  MoveC 1133 to (433.16, 156.25, -8.35) mm, rotated rx 180 ry 0 rz -179 deg; joints [11.722, -45.324, 75.106, 22.673, -31.807, -19.546] to (420.46, 168.95, -8.35) mm, rotated rx -180 ry 0 rz -179 deg; joints [11.384, -46.351, 76.909, 21.605, -32.417, -18.486]
  MoveL 1134 to (395.06, 168.95, -8.35) mm, rotated rx -180 ry 0 rz -179 deg; joints [11.539, -48.04, 79.855, 21.171, -33.635, -17.872]
  MoveL 1135 to (318.86, 168.95, -8.35) mm, rotated rx -180 ry 0 rz -179 deg; joints [12.033, -52.857, 88.085, 20.282, -36.974, -16.448]
  MoveC 1136 to (306.16, 156.25, -8.35) mm, rotated rx -180 ry 0 rz -179 deg; joints [12.565, -53.476, 89.123, 20.928, -37.518, -16.874] to (293.46, 168.95, -8.35) mm, rotated rx -180 ry 0 rz -179 deg; joints [12.208, -54.397, 90.66, 20.092, -37.994, -16.081]
  MoveL 1137 to (191.86, 168.95, -8.35) mm, rotated rx -180 ry 0 rz -179 deg; joints [12.967, -60.337, 100.305, 19.72, -41.681, -14.987]
  MoveC 1138 to (179.16, 156.25, -8.35) mm, rotated rx 180 ry 0 rz -179 deg; joints [13.549, -60.904, 101.2, 20.435, -42.142, -15.444] to (166.46, 168.95, -8.35) mm, rotated rx 180 ry 0 rz -179 deg; joints [13.172, -61.782, 102.578, 19.708, -42.513, -14.791]
  MoveL 1139 to (90.26, 168.95, -8.35) mm, rotated rx -180 ry 0 rz -179 deg; joints [13.833, -66.063, 109.12, 19.833, -44.808, -14.353]
  MoveL 1140 to (64.86, 168.95, -8.35) mm, rotated rx -180 ry 0 rz -179 deg; joints [14.069, -67.479, 111.218, 19.925, -45.508, -14.253]
  MoveC 1141 to (61.14, 159.97, -8.35) mm, rotated rx -180 ry 0 rz -179 deg; joints [14.471, -67.568, 111.349, 20.456, -45.647, -14.615] to (52.16, 156.25, -8.35) mm, rotated rx 180 ry 0 rz -179 deg; joints [14.712, -68.017, 112.007, 20.709, -45.903, -14.739]
  MoveL 1142 to (52.16, 156.25, -8.35) mm, rotated rx 180 ry 0 rz -179 deg; joints [14.712, -68.017, 112.007, 20.709, -45.903, -14.739]
  MoveC 1143 to (43.18, 159.97, -8.35) mm, rotated rx -180 ry 0 rz -179 deg; joints [14.649, -68.566, 112.806, 20.539, -46.122, -14.558] to (39.46, 168.95, -8.35) mm, rotated rx -180 ry 0 rz -179 deg; joints [14.314, -68.892, 113.279, 20.041, -46.176, -14.176]
  MoveL 1144 to (14.06, 168.95, -8.35) mm, rotated rx 180 ry 0 rz -179 deg; joints [14.568, -70.305, 115.303, 20.181, -46.812, -14.12]
  MoveL 1145 to (14.06, 16.55, -8.35) mm, rotated rx 180 ry 0 rz -179 deg; joints [20.81, -67.799, 111.688, 28.732, -47.649, -20.27]
  MoveL 1146 to (19.05, 16.55, -8.35) mm, rotated rx -180 ry 0 rz -179 deg; joints [20.739, -67.53, 111.295, 28.697, -47.515, -20.291]
  MoveC 1147 to (19.49, 16.36, -8.35) mm, rotated rx -180 ry 0 rz -179 deg; joints [20.74, -67.503, 111.254, 28.704, -47.504, -20.3] to (19.68, 15.92, -8.35) mm, rotated rx -180 ry 0 rz -179 deg; joints [20.755, -67.484, 111.226, 28.727, -47.501, -20.319]
  MoveL 1148 to (19.68, 15.28, -8.35) mm, rotated rx -180 ry 0 rz -179 deg; joints [20.78, -67.472, 111.208, 28.762, -47.505, -20.344]
  MoveC 1149 to (19.68, 14.83, -8.16) mm, rotated rx 180 ry 0 rz -179 deg; joints [20.798, -67.47, 111.191, 28.791, -47.497, -20.37] to (19.68, 14.65, -7.72) mm, rotated rx 180 ry 0 rz -179 deg; joints [20.805, -67.484, 111.173, 28.814, -47.473, -20.396]
  Set speed (500.0 mm/s)
  MoveL 1150 to (19.68, 14.65, 6) mm, rotated rx -180 ry 0 rz -179 deg; joints [20.805, -68, 110.8, 29.215, -46.695, -20.985]
  MoveL 1151 to (12.15, -16.75, 6) mm, rotated rx -180 ry 0 rz -179 deg; joints [22.145, -67.773, 110.469, 30.97, -47.099, -22.222]
  Set speed (25.4 mm/s)
  MoveL 1152 to (12.15, -16.75, -4.37) mm, rotated rx 180 ry 0 rz -179 deg; joints [22.145, -67.386, 110.753, 30.654, -47.675, -21.756]
  MoveC 1153 to (12.34, -16.75, -4.81) mm, rotated rx -180 ry 0 rz -179 deg; joints [22.142, -67.359, 110.75, 30.639, -47.694, -21.736] to (12.79, -16.75, -5) mm, rotated rx -180 ry 0 rz -179 deg; joints [22.135, -67.328, 110.72, 30.63, -47.693, -21.73]
  Set speed (50.8 mm/s)
  MoveL 1154 to (13.42, -16.75, -5) mm, rotated rx -180 ry 0 rz -179 deg; joints [22.126, -67.294, 110.67, 30.626, -47.675, -21.733]
  MoveC 1155 to (13.87, -16.94, -5) mm, rotated rx -180 ry 0 rz -179 deg; joints [22.126, -67.266, 110.629, 30.633, -47.664, -21.743] to (14.06, -17.39, -5) mm, rotated rx 180 ry 0 rz -179 deg; joints [22.141, -67.247, 110.601, 30.655, -47.662, -21.761]
  MoveL 1156 to (14.06, -169.79, -5) mm, rotated rx -180 ry 0 rz -179 deg; joints [27.82, -63.684, 105.249, 38.496, -48.568, -27.757]
  MoveL 1157 to (471.26, -169.79, -5) mm, rotated rx -180 ry 0 rz -179 deg; joints [21.439, -35.651, 57.394, 46.669, -30.164, -42.505]
  MoveL 1158 to (471.26, -17.39, -5) mm, rotated rx 180 ry 0 rz -179 deg; joints [16.91, -39.664, 64.74, 35.652, -29.935, -31.866]
  MoveL 1159 to (445.86, -17.39, -5) mm, rotated rx -180 ry 0 rz -179 deg; joints [17.133, -41.565, 68.171, 34.541, -31.303, -30.461]
  MoveC 1160 to (433.16, -30.09, -5) mm, rotated rx -180 ry 0 rz -179 deg; joints [17.641, -42.214, 69.335, 34.898, -31.985, -30.611] to (420.46, -17.39, -5) mm, rotated rx -180 ry 0 rz -179 deg; joints [17.363, -43.381, 71.42, 33.631, -32.604, -29.264]
  MoveL 1161 to (395.06, -17.39, -5) mm, rotated rx 180 ry 0 rz -179 deg; joints [17.599, -45.128, 74.514, 32.88, -33.845, -28.231]
  MoveL 1162 to (318.86, -17.39, -5) mm, rotated rx 180 ry 0 rz -179 deg; joints [18.35, -50.044, 83.06, 31.33, -37.261, -25.849]
  MoveC 1163 to (306.16, -30.09, -5) mm, rotated rx 180 ry 0 rz -179 deg; joints [18.901, -50.578, 83.972, 31.885, -37.825, -26.168] to (293.46, -17.39, -5) mm, rotated rx 180 ry 0 rz -179 deg; joints [18.614, -51.599, 85.709, 30.99, -38.311, -25.234]
  MoveL 1164 to (191.86, -17.39, -5) mm, rotated rx -180 ry 0 rz -179 deg; joints [19.757, -57.528, 95.542, 30.252, -42.142, -23.386]
  MoveC 1165 to (179.16, -30.09, -5) mm, rotated rx 180 ry 0 rz -179 deg; joints [20.359, -57.996, 96.299, 30.909, -42.631, -23.772] to (166.46, -17.39, -5) mm, rotated rx -180 ry 0 rz -179 deg; joints [20.065, -58.955, 97.84, 30.193, -43.017, -23.046]
  MoveL 1166 to (90.26, -17.39, -5) mm, rotated rx -180 ry 0 rz -179 deg; joints [21.052, -63.146, 104.423, 30.261, -45.463, -22.255]
  MoveL 1167 to (64.86, -17.39, -5) mm, rotated rx -180 ry 0 rz -179 deg; joints [21.403, -64.521, 106.524, 30.358, -46.223, -22.059]
  MoveC 1168 to (61.14, -26.37, -5) mm, rotated rx -180 ry 0 rz -179 deg; joints [21.794, -64.539, 106.552, 30.855, -46.379, -22.399] to (52.16, -30.09, -5) mm, rotated rx -180 ry 0 rz -179 deg; joints [22.064, -64.945, 107.167, 31.097, -46.661, -22.487]
  MoveL 1169 to (52.16, -30.09, -5) mm, rotated rx -180 ry 0 rz -179 deg; joints [22.064, -64.945, 107.167, 31.097, -46.661, -22.487]
  MoveC 1170 to (43.18, -26.37, -5) mm, rotated rx -180 ry 0 rz -179 deg; joints [22.054, -65.503, 108.008, 30.947, -46.9, -22.279] to (39.46, -17.39, -5) mm, rotated rx -180 ry 0 rz -179 deg; joints [21.766, -65.887, 108.583, 30.49, -46.955, -21.895]
  MoveL 1171 to (14.06, -17.39, -5) mm, rotated rx -180 ry 0 rz -179 deg; joints [22.141, -67.247, 110.601, 30.655, -47.662, -21.761]
  MoveC 1172 to (13.61, -17.2, -5) mm, rotated rx -180 ry 0 rz -179 deg; joints [22.14, -67.275, 110.642, 30.648, -47.673, -21.752] to (13.42, -16.75, -5) mm, rotated rx -180 ry 0 rz -179 deg; joints [22.126, -67.294, 110.67, 30.626, -47.675, -21.733]
  MoveL 1173 to (13.42, -16.12, -5) mm, rotated rx -180 ry 0 rz -179 deg; joints [22.101, -67.307, 110.689, 30.592, -47.671, -21.708]
  MoveC 1174 to (13.42, -15.67, -4.81) mm, rotated rx -180 ry 0 rz -179 deg; joints [22.084, -67.323, 110.698, 30.574, -47.658, -21.698] to (13.42, -15.48, -4.37) mm, rotated rx -180 ry 0 rz -179 deg; joints [22.076, -67.344, 110.692, 30.577, -47.632, -21.711]
  Set speed (500.0 mm/s)
  MoveL 1175 to (13.42, -15.48, 5) mm, rotated rx -180 ry 0 rz -179 deg; joints [22.076, -67.694, 110.436, 30.862, -47.112, -22.131]
  MoveL 1176 to (12.15, -16.75, 5) mm, rotated rx -180 ry 0 rz -179 deg; joints [22.145, -67.736, 110.497, 30.939, -47.154, -22.177]
  Set speed (25.4 mm/s)
  MoveL 1177 to (12.15, -16.75, 1) mm, rotated rx -180 ry 0 rz -179 deg; joints [22.145, -67.587, 110.607, 30.816, -47.376, -21.996]
  MoveL 1178 to (12.15, -16.75, -7.71) mm, rotated rx 180 ry 0 rz -179 deg; joints [22.145, -67.259, 110.843, 30.554, -47.861, -21.607]
  MoveC 1179 to (12.34, -16.75, -8.16) mm, rotated rx -180 ry 0 rz -179 deg; joints [22.142, -67.232, 110.84, 30.539, -47.881, -21.588] to (12.79, -16.75, -8.35) mm, rotated rx 180 ry 0 rz -179 deg; joints [22.135, -67.201, 110.81, 30.531, -47.879, -21.582]
  Set speed (50.8 mm/s)
  MoveL 1180 to (13.42, -16.75, -8.35) mm, rotated rx -180 ry 0 rz -179 deg; joints [22.126, -67.167, 110.76, 30.526, -47.861, -21.584]
  MoveC 1181 to (13.87, -16.94, -8.35) mm, rotated rx 180 ry 0 rz -179 deg; joints [22.126, -67.139, 110.719, 30.533, -47.85, -21.594] to (14.06, -17.39, -8.35) mm, rotated rx -180 ry 0 rz -179 deg; joints [22.141, -67.12, 110.69, 30.555, -47.848, -21.613]
  MoveL 1182 to (14.06, -169.79, -8.35) mm, rotated rx 180 ry 0 rz -179 deg; joints [27.82, -63.565, 105.338, 38.383, -48.731, -27.585]
  MoveL 1183 to (471.26, -169.79, -8.35) mm, rotated rx -180 ry 0 rz -179 deg; joints [21.439, -35.589, 57.514, 46.442, -30.289, -42.242]
  MoveL 1184 to (471.26, -17.39, -8.35) mm, rotated rx -180 ry 0 rz -179 deg; joints [16.91, -39.592, 64.848, 35.471, -30.082, -31.656]
  MoveL 1185 to (445.86, -17.39, -8.35) mm, rotated rx -180 ry 0 rz -179 deg; joints [17.133, -41.488, 68.274, 34.374, -31.452, -30.266]
  MoveC 1186 to (433.16, -30.09, -8.35) mm, rotated rx -180 ry 0 rz -179 deg; joints [17.641, -42.136, 69.438, 34.734, -32.133, -30.418] to (420.46, -17.39, -8.35) mm, rotated rx -180 ry 0 rz -179 deg; joints [17.363, -43.301, 71.52, 33.475, -32.754, -29.08]
  MoveL 1187 to (395.06, -17.39, -8.35) mm, rotated rx -180 ry 0 rz -179 deg; joints [17.599, -45.045, 74.612, 32.734, -33.997, -28.056]
  MoveL 1188 to (318.86, -17.39, -8.35) mm, rotated rx 180 ry 0 rz -179 deg; joints [18.35, -49.952, 83.152, 31.204, -37.419, -25.691]
  MoveC 1189 to (306.16, -30.09, -8.35) mm, rotated rx -180 ry 0 rz -179 deg; joints [18.901, -50.485, 84.064, 31.759, -37.982, -26.009] to (293.46, -17.39, -8.35) mm, rotated rx 180 ry 0 rz -179 deg; joints [18.614, -51.504, 85.799, 30.869, -38.471, -25.08]
  MoveL 1190 to (191.86, -17.39, -8.35) mm, rotated rx 180 ry 0 rz -179 deg; joints [19.757, -57.421, 95.63, 30.144, -42.31, -23.24]
  MoveC 1191 to (179.16, -30.09, -8.35) mm, rotated rx -180 ry 0 rz -179 deg; joints [20.359, -57.889, 96.387, 30.8, -42.799, -23.624] to (166.46, -17.39, -8.35) mm, rotated rx -180 ry 0 rz -179 deg; joints [20.065, -58.846, 97.928, 30.087, -43.187, -22.901]
  MoveL 1192 to (90.26, -17.39, -8.35) mm, rotated rx 180 ry 0 rz -179 deg; joints [21.052, -63.028, 104.512, 30.16, -45.642, -22.11]
  MoveL 1193 to (64.86, -17.39, -8.35) mm, rotated rx 180 ry 0 rz -179 deg; joints [21.403, -64.4, 106.613, 30.257, -46.404, -21.913]
  MoveC 1194 to (61.14, -26.37, -8.35) mm, rotated rx -180 ry 0 rz -179 deg; joints [21.794, -64.418, 106.641, 30.753, -46.559, -22.251] to (52.16, -30.09, -8.35) mm, rotated rx -180 ry 0 rz -179 deg; joints [22.064, -64.823, 107.256, 30.995, -46.841, -22.339]
  MoveL 1195 to (52.16, -30.09, -8.35) mm, rotated rx 180 ry 0 rz -179 deg; joints [22.064, -64.823, 107.256, 30.995, -46.841, -22.339]
  MoveC 1196 to (43.18, -26.37, -8.35) mm, rotated rx 180 ry 0 rz -179 deg; joints [22.054, -65.381, 108.097, 30.846, -47.081, -22.13] to (39.46, -17.39, -8.35) mm, rotated rx -180 ry 0 rz -179 deg; joints [21.766, -65.763, 108.672, 30.39, -47.139, -21.748]
  MoveL 1197 to (14.06, -17.39, -8.35) mm, rotated rx -180 ry 0 rz -179 deg; joints [22.141, -67.12, 110.69, 30.555, -47.848, -21.613]
  MoveC 1198 to (13.61, -17.2, -8.35) mm, rotated rx 180 ry 0 rz -179 deg; joints [22.14, -67.148, 110.731, 30.549, -47.859, -21.603] to (13.42, -16.75, -8.35) mm, rotated rx -180 ry 0 rz -179 deg; joints [22.126, -67.167, 110.76, 30.526, -47.861, -21.584]
  MoveL 1199 to (13.42, -16.12, -8.35) mm, rotated rx 180 ry 0 rz -179 deg; joints [22.101, -67.18, 110.779, 30.492, -47.858, -21.559]
  MoveC 1200 to (13.42, -15.67, -8.16) mm, rotated rx -180 ry 0 rz -179 deg; joints [22.084, -67.196, 110.788, 30.474, -47.845, -21.55] to (13.42, -15.48, -7.72) mm, rotated rx -180 ry 0 rz -179 deg; joints [22.076, -67.217, 110.781, 30.477, -47.819, -21.562]
  Set speed (500.0 mm/s)
  MoveL 1201 to (13.42, -15.48, 6) mm, rotated rx -180 ry 0 rz -179 deg; joints [22.076, -67.731, 110.408, 30.893, -47.056, -22.177]
  MoveL 1202 to (-18.41, -15.48, 6) mm, rotated rx 180 ry 0 rz -179 deg; joints [22.565, -69.442, 112.879, 31.147, -47.892, -22.06]
  Set speed (25.4 mm/s)
  MoveL 1203 to (-18.41, -15.48, -4.36) mm, rotated rx 180 ry 0 rz -179 deg; joints [22.565, -69.043, 113.165, 30.832, -48.478, -21.587]
  MoveC 1204 to (-18.41, -15.67, -4.81) mm, rotated rx -180 ry 0 rz -179 deg; joints [22.572, -69.022, 113.172, 30.828, -48.505, -21.574] to (-18.41, -16.12, -5) mm, rotated rx -180 ry 0 rz -179 deg; joints [22.59, -69.005, 113.163, 30.847, -48.518, -21.583]
  Set speed (50.8 mm/s)
  MoveL 1205 to (-18.41, -16.75, -5) mm, rotated rx -180 ry 0 rz -179 deg; joints [22.615, -68.992, 113.144, 30.88, -48.523, -21.608]
  MoveC 1206 to (-18.6, -17.2, -5) mm, rotated rx -180 ry 0 rz -179 deg; joints [22.636, -68.992, 113.145, 30.906, -48.53, -21.625] to (-19.05, -17.39, -5) mm, rotated rx -180 ry 0 rz -179 deg; joints [22.65, -69.012, 113.174, 30.92, -48.543, -21.631]
  MoveL 1207 to (-39.46, -17.39, -5) mm, rotated rx -180 ry 0 rz -179 deg; joints [22.976, -70.099, 114.729, 31.111, -49.065, -21.574]
  MoveC 1208 to (-52.16, -30.09, -5) mm, rotated rx 180 ry 0 rz -179 deg; joints [23.694, -70.496, 115.292, 31.917, -49.474, -22.034] to (-64.86, -17.39, -5) mm, rotated rx -180 ry 0 rz -179 deg; joints [23.394, -71.449, 116.633, 31.377, -49.692, -21.53]
  MoveL 1209 to (-90.26, -17.39, -5) mm, rotated rx -180 ry 0 rz -179 deg; joints [23.828, -72.8, 118.503, 31.676, -50.294, -21.514]
  MoveL 1210 to (-166.46, -17.39, -5) mm, rotated rx 180 ry 0 rz -179 deg; joints [25.231, -76.869, 123.921, 32.772, -51.951, -21.642]
  MoveC 1211 to (-179.16, -30.09, -5) mm, rotated rx 180 ry 0 rz -179 deg; joints [26.031, -77.238, 124.395, 33.668, -52.338, -22.146] to (-191.86, -17.39, -5) mm, rotated rx 180 ry 0 rz -179 deg; joints [25.735, -78.236, 125.666, 33.205, -52.454, -21.745]
  MoveL 1212 to (-293.46, -17.39, -5) mm, rotated rx -180 ry 0 rz -179 deg; joints [27.963, -83.794, 132.347, 35.308, -54.222, -22.493]
  MoveC 1213 to (-306.16, -30.09, -5) mm, rotated rx 180 ry 0 rz -179 deg; joints [28.862, -84.133, 132.733, 36.308, -54.608, -23.053] to (-318.86, -17.39, -5) mm, rotated rx -180 ry 0 rz -179 deg; joints [28.579, -85.214, 133.944, 35.933, -54.604, -22.773]
  MoveL 1214 to (-395.06, -17.39, -5) mm, rotated rx -180 ry 0 rz -179 deg; joints [30.593, -89.571, 138.561, 38.079, -55.608, -23.872]
  MoveL 1215 to (-420.46, -17.39, -5) mm, rotated rx -180 ry 0 rz -179 deg; joints [31.325, -91.061, 140.04, 38.892, -55.899, -24.335]
  MoveC 1216 to (-433.16, -30.09, -5) mm, rotated rx 180 ry 0 rz -179 deg; joints [32.344, -91.362, 140.333, 40.011, -56.317, -24.964] to (-445.86, -17.39, -5) mm, rotated rx 180 ry 0 rz -179 deg; joints [32.091, -92.572, 141.489, 39.758, -56.169, -24.852]
  MoveL 1217 to (-471.26, -17.39, -5) mm, rotated rx 180 ry 0 rz -179 deg; joints [32.892, -94.107, 142.906, 40.68, -56.42, -25.427]
  MoveL 1218 to (-471.26, -169.79, -5) mm, rotated rx 180 ry 0 rz -179 deg; joints [40.129, -88.033, 136.981, 48.184, -59.858, -29.305]
  MoveL 1219 to (-14.06, -169.79, -5) mm, rotated rx -180 ry 0 rz -179 deg; joints [28.334, -65.125, 107.439, 38.694, -49.392, -27.535]
  MoveL 1220 to (-14.06, -17.39, -5) mm, rotated rx 180 ry 0 rz -179 deg; joints [22.572, -68.747, 112.79, 30.877, -48.413, -21.647]
  MoveL 1221 to (-19.05, -17.39, -5) mm, rotated rx -180 ry 0 rz -179 deg; joints [22.65, -69.012, 113.174, 30.92, -48.543, -21.631]
  MoveC 1222 to (-19.49, -17.2, -5) mm, rotated rx 180 ry 0 rz -179 deg; joints [22.65, -69.04, 113.214, 30.914, -48.554, -21.622] to (-19.68, -16.75, -5) mm, rotated rx -180 ry 0 rz -179 deg; joints [22.635, -69.06, 113.242, 30.892, -48.556, -21.604]
  MoveL 1223 to (-19.68, -16.12, -5) mm, rotated rx 180 ry 0 rz -179 deg; joints [22.61, -69.073, 113.261, 30.858, -48.551, -21.579]
  MoveC 1224 to (-19.68, -15.67, -4.81) mm, rotated rx -180 ry 0 rz -179 deg; joints [22.592, -69.09, 113.27, 30.839, -48.538, -21.57] to (-19.68, -15.48, -4.37) mm, rotated rx -180 ry 0 rz -179 deg; joints [22.584, -69.111, 113.263, 30.843, -48.511, -21.583]
  Set speed (500.0 mm/s)
  MoveL 1225 to (-19.68, -15.48, 5) mm, rotated rx -180 ry 0 rz -179 deg; joints [22.584, -69.472, 113.005, 31.127, -47.981, -22.01]
  MoveL 1226 to (-18.41, -15.48, 5) mm, rotated rx -180 ry 0 rz -179 deg; joints [22.565, -69.404, 112.907, 31.116, -47.948, -22.014]
  Set speed (25.4 mm/s)
  MoveL 1227 to (-18.41, -15.48, 1) mm, rotated rx -180 ry 0 rz -179 deg; joints [22.565, -69.25, 113.019, 30.994, -48.175, -21.831]
  MoveL 1228 to (-18.41, -15.48, -7.72) mm, rotated rx 180 ry 0 rz -179 deg; joints [22.565, -68.913, 113.256, 30.732, -48.668, -21.436]
  MoveC 1229 to (-18.41, -15.67, -8.16) mm, rotated rx -180 ry 0 rz -179 deg; joints [22.572, -68.891, 113.263, 30.728, -48.695, -21.423] to (-18.41, -16.12, -8.35) mm, rotated rx 180 ry 0 rz -179 deg; joints [22.59, -68.875, 113.254, 30.747, -48.708, -21.432]
  Set speed (50.8 mm/s)
  MoveL 1230 to (-18.41, -16.75, -8.35) mm, rotated rx -180 ry 0 rz -179 deg; joints [22.615, -68.861, 113.235, 30.781, -48.712, -21.457]
  MoveC 1231 to (-18.6, -17.2, -8.35) mm, rotated rx 180 ry 0 rz -179 deg; joints [22.636, -68.862, 113.235, 30.806, -48.72, -21.474] to (-19.05, -17.39, -8.35) mm, rotated rx 180 ry 0 rz -179 deg; joints [22.65, -68.882, 113.264, 30.82, -48.733, -21.479]
  MoveL 1232 to (-39.46, -17.39, -8.35) mm, rotated rx 180 ry 0 rz -179 deg; joints [22.976, -69.966, 114.82, 31.011, -49.257, -21.421]
  MoveC 1233 to (-52.16, -30.09, -8.35) mm, rotated rx 180 ry 0 rz -179 deg; joints [23.694, -70.362, 115.384, 31.815, -49.665, -21.878] to (-64.86, -17.39, -8.35) mm, rotated rx -180 ry 0 rz -179 deg; joints [23.394, -71.313, 116.725, 31.277, -49.887, -21.375]
  MoveL 1234 to (-90.26, -17.39, -8.35) mm, rotated rx -180 ry 0 rz -179 deg; joints [23.828, -72.661, 118.596, 31.576, -50.492, -21.356]
  MoveL 1235 to (-166.46, -17.39, -8.35) mm, rotated rx 180 ry 0 rz -179 deg; joints [25.231, -76.72, 124.018, 32.668, -52.158, -21.473]
  MoveC 1236 to (-179.16, -30.09, -8.35) mm, rotated rx 180 ry 0 rz -179 deg; joints [26.031, -77.088, 124.492, 33.563, -52.544, -21.974] to (-191.86, -17.39, -8.35) mm, rotated rx -180 ry 0 rz -179 deg; joints [25.735, -78.083, 125.763, 33.1, -52.664, -21.572]
  MoveL 1237 to (-293.46, -17.39, -8.35) mm, rotated rx 180 ry 0 rz -179 deg; joints [27.963, -83.627, 132.451, 35.196, -54.443, -22.301]
  MoveC 1238 to (-306.16, -30.09, -8.35) mm, rotated rx 180 ry 0 rz -179 deg; joints [28.862, -83.965, 132.837, 36.194, -54.828, -22.856] to (-318.86, -17.39, -8.35) mm, rotated rx -180 ry 0 rz -179 deg; joints [28.579, -85.043, 134.05, 35.818, -54.828, -22.574]
  MoveL 1239 to (-395.06, -17.39, -8.35) mm, rotated rx -180 ry 0 rz -179 deg; joints [30.593, -89.388, 138.674, 37.955, -55.841, -23.653]
  MoveL 1240 to (-420.46, -17.39, -8.35) mm, rotated rx -180 ry 0 rz -179 deg; joints [31.325, -90.874, 140.155, 38.765, -56.134, -24.108]
  MoveC 1241 to (-433.16, -30.09, -8.35) mm, rotated rx -180 ry 0 rz -179 deg; joints [32.344, -91.175, 140.449, 39.882, -56.549, -24.731] to (-445.86, -17.39, -8.35) mm, rotated rx 180 ry 0 rz -179 deg; joints [32.091, -92.382, 141.607, 39.627, -56.406, -24.616]
  MoveL 1242 to (-471.26, -17.39, -8.35) mm, rotated rx -180 ry 0 rz -179 deg; joints [32.892, -93.913, 143.027, 40.545, -56.658, -25.182]
  MoveL 1243 to (-471.26, -169.79, -8.35) mm, rotated rx 180 ry 0 rz -179 deg; joints [40.129, -87.855, 137.091, 48.059, -60.051, -29.057]
  MoveL 1244 to (-14.06, -169.79, -8.35) mm, rotated rx -180 ry 0 rz -179 deg; joints [28.334, -65.003, 107.528, 38.582, -49.557, -27.362]
  MoveL 1245 to (-14.06, -17.39, -8.35) mm, rotated rx -180 ry 0 rz -179 deg; joints [22.572, -68.617, 112.88, 30.777, -48.602, -21.496]
  MoveL 1246 to (-19.05, -17.39, -8.35) mm, rotated rx 180 ry 0 rz -179 deg; joints [22.65, -68.882, 113.264, 30.82, -48.733, -21.479]
  MoveC 1247 to (-19.49, -17.2, -8.35) mm, rotated rx -180 ry 0 rz -179 deg; joints [22.65, -68.91, 113.304, 30.814, -48.744, -21.471] to (-19.68, -16.75, -8.35) mm, rotated rx 180 ry 0 rz -179 deg; joints [22.635, -68.929, 113.332, 30.792, -48.745, -21.453]
  MoveL 1248 to (-19.68, -16.12, -8.35) mm, rotated rx -180 ry 0 rz -179 deg; joints [22.61, -68.942, 113.351, 30.758, -48.741, -21.428]
  MoveC 1249 to (-19.68, -15.67, -8.16) mm, rotated rx -180 ry 0 rz -179 deg; joints [22.592, -68.959, 113.36, 30.74, -48.728, -21.419] to (-19.68, -15.48, -7.72) mm, rotated rx 180 ry 0 rz -179 deg; joints [22.584, -68.98, 113.354, 30.743, -48.701, -21.432]
  Set speed (500.0 mm/s)
  MoveL 1250 to (-19.68, -15.48, 6) mm, rotated rx -180 ry 0 rz -179 deg; joints [22.584, -69.51, 112.977, 31.158, -47.924, -22.056]
  MoveL 1251 to (-13.42, -196.51, 6) mm, rotated rx 180 ry 0 rz -179 deg; joints [29.278, -64.766, 106.007, 40.38, -49.013, -29.154]
  Set speed (25.4 mm/s)
  MoveL 1252 to (-13.42, -196.52, -4.36) mm, rotated rx -180 ry 0 rz -179 deg; joints [29.278, -64.399, 106.288, 40.02, -49.508, -28.602]
  MoveC 1253 to (-13.42, -196.7, -4.81) mm, rotated rx -180 ry 0 rz -179 deg; joints [29.284, -64.377, 106.292, 40.014, -49.53, -28.585] to (-13.42, -197.15, -5) mm, rotated rx 180 ry 0 rz -179 deg; joints [29.3, -64.358, 106.278, 40.029, -49.542, -28.593]
  Set speed (50.8 mm/s)
  MoveL 1254 to (-13.42, -197.78, -5) mm, rotated rx 180 ry 0 rz -179 deg; joints [29.323, -64.341, 106.252, 40.06, -49.546, -28.617]
  MoveC 1255 to (-13.61, -198.23, -5) mm, rotated rx -180 ry 0 rz -179 deg; joints [29.342, -64.338, 106.247, 40.084, -49.554, -28.633] to (-14.06, -198.42, -5) mm, rotated rx 180 ry 0 rz -179 deg; joints [29.357, -64.356, 106.274, 40.096, -49.568, -28.636]
  MoveL 1256 to (-39.46, -198.42, -5) mm, rotated rx 180 ry 0 rz -179 deg; joints [29.85, -65.638, 108.21, 40.307, -50.303, -28.449]
  MoveC 1257 to (-52.16, -211.12, -5) mm, rotated rx -180 ry 0 rz -179 deg; joints [30.557, -65.918, 108.63, 41.036, -50.748, -28.843] to (-64.86, -198.42, -5) mm, rotated rx 180 ry 0 rz -179 deg; joints [30.359, -66.911, 110.105, 40.555, -51.019, -28.294]
  MoveL 1258 to (-90.26, -198.42, -5) mm, rotated rx -180 ry 0 rz -179 deg; joints [30.884, -68.176, 111.961, 40.839, -51.715, -28.171]
  MoveL 1259 to (-166.46, -198.42, -5) mm, rotated rx -180 ry 0 rz -179 deg; joints [32.567, -71.935, 117.309, 41.906, -53.7, -27.981]
  MoveC 1260 to (-179.16, -211.12, -5) mm, rotated rx -180 ry 0 rz -179 deg; joints [33.344, -72.168, 117.633, 42.709, -54.133, -28.405] to (-191.86, -198.42, -5) mm, rotated rx -180 ry 0 rz -179 deg; joints [33.166, -73.179, 119.022, 42.332, -54.328, -27.978]
  MoveL 1261 to (-293.46, -198.42, -5) mm, rotated rx -180 ry 0 rz -179 deg; joints [35.779, -78.138, 125.542, 44.391, -56.695, -28.26]
  MoveC 1262 to (-306.16, -211.12, -5) mm, rotated rx 180 ry 0 rz -179 deg; joints [36.635, -78.319, 125.771, 45.267, -57.137, -28.71] to (-318.86, -198.42, -5) mm, rotated rx 180 ry 0 rz -179 deg; joints [36.491, -79.376, 127.091, 44.997, -57.254, -28.407]
  MoveL 1263 to (-395.06, -198.42, -5) mm, rotated rx -180 ry 0 rz -179 deg; joints [38.787, -83.099, 131.548, 47.039, -58.868, -29.039]
  MoveL 1264 to (-420.46, -198.42, -5) mm, rotated rx 180 ry 0 rz -179 deg; joints [39.609, -84.344, 132.971, 47.798, -59.389, -29.316]
  MoveC 1265 to (-433.16, -211.12, -5) mm, rotated rx 180 ry 0 rz -179 deg; joints [40.554, -84.46, 133.102, 48.744, -59.865, -29.784] to (-445.86, -198.42, -5) mm, rotated rx -180 ry 0 rz -179 deg; joints [40.462, -85.591, 134.361, 48.596, -59.904, -29.627]
  MoveL 1266 to (-471.26, -198.42, -5) mm, rotated rx 180 ry 0 rz -179 deg; joints [41.347, -86.841, 135.719, 49.434, -60.414, -29.973]
  MoveL 1267 to (-471.26, -350.82, -5) mm, rotated rx -180 ry 0 rz -179 deg; joints [47.144, -80.326, 128.256, 55.442, -62.888, -33.491]
  MoveL 1268 to (-14.06, -350.82, -5) mm, rotated rx -180 ry 0 rz -179 deg; joints [34.476, -59.803, 99.193, 47.256, -50.424, -34.581]
  MoveL 1269 to (-14.06, -198.42, -5) mm, rotated rx 180 ry 0 rz -179 deg; joints [29.357, -64.356, 106.274, 40.096, -49.568, -28.636]
  MoveC 1270 to (-13.87, -197.97, -5) mm, rotated rx -180 ry 0 rz -179 deg; joints [29.338, -64.359, 106.279, 40.073, -49.56, -28.621] to (-13.42, -197.78, -5) mm, rotated rx 180 ry 0 rz -179 deg; joints [29.323, -64.341, 106.252, 40.06, -49.546, -28.617]
  MoveL 1271 to (-12.79, -197.78, -5) mm, rotated rx -180 ry 0 rz -179 deg; joints [29.31, -64.309, 106.203, 40.056, -49.527, -28.622]
  MoveC 1272 to (-12.34, -197.78, -4.81) mm, rotated rx 180 ry 0 rz -179 deg; joints [29.302, -64.293, 106.163, 40.059, -49.505, -28.636] to (-12.15, -197.79, -4.37) mm, rotated rx 180 ry 0 rz -179 deg; joints [29.298, -64.299, 106.137, 40.073, -49.478, -28.661]
  Set speed (500.0 mm/s)
  MoveL 1273 to (-12.15, -197.78, 5) mm, rotated rx 180 ry 0 rz -179 deg; joints [29.298, -64.631, 105.884, 40.398, -49.032, -29.159]
  MoveL 1274 to (-13.42, -196.52, 5) mm, rotated rx 180 ry 0 rz -179 deg; joints [29.278, -64.731, 106.035, 40.345, -49.061, -29.1]
  Set speed (25.4 mm/s)
  MoveL 1275 to (-13.42, -196.51, 1) mm, rotated rx -180 ry 0 rz -179 deg; joints [29.278, -64.59, 106.144, 40.205, -49.251, -28.886]
  MoveL 1276 to (-13.42, -196.51, -7.72) mm, rotated rx 180 ry 0 rz -179 deg; joints [29.278, -64.278, 106.376, 39.906, -49.668, -28.425]
  MoveC 1277 to (-13.42, -196.7, -8.16) mm, rotated rx -180 ry 0 rz -179 deg; joints [29.284, -64.257, 106.38, 39.9, -49.691, -28.409] to (-13.42, -197.15, -8.35) mm, rotated rx 180 ry 0 rz -179 deg; joints [29.3, -64.238, 106.367, 39.915, -49.702, -28.416]
  Set speed (50.8 mm/s)
  MoveL 1278 to (-13.42, -197.78, -8.35) mm, rotated rx -180 ry 0 rz -179 deg; joints [29.323, -64.221, 106.34, 39.946, -49.706, -28.441]
  MoveC 1279 to (-13.61, -198.23, -8.35) mm, rotated rx 180 ry 0 rz -179 deg; joints [29.342, -64.218, 106.336, 39.969, -49.714, -28.457] to (-14.06, -198.42, -8.35) mm, rotated rx -180 ry 0 rz -179 deg; joints [29.357, -64.236, 106.363, 39.982, -49.728, -28.46]
  MoveL 1280 to (-39.46, -198.42, -8.35) mm, rotated rx -180 ry 0 rz -179 deg; joints [29.85, -65.515, 108.299, 40.193, -50.465, -28.271]
  MoveC 1281 to (-52.16, -211.12, -8.35) mm, rotated rx 180 ry 0 rz -179 deg; joints [30.557, -65.795, 108.719, 40.922, -50.909, -28.663] to (-64.86, -198.42, -8.35) mm, rotated rx 180 ry 0 rz -179 deg; joints [30.359, -66.785, 110.194, 40.442, -51.182, -28.115]
  MoveL 1282 to (-90.26, -198.42, -8.35) mm, rotated rx -180 ry 0 rz -179 deg; joints [30.884, -68.047, 112.051, 40.727, -51.881, -27.989]
  MoveL 1283 to (-166.46, -198.42, -8.35) mm, rotated rx -180 ry 0 rz -179 deg; joints [32.567, -71.798, 117.402, 41.794, -53.871, -27.792]
  MoveC 1284 to (-179.16, -211.12, -8.35) mm, rotated rx -180 ry 0 rz -179 deg; joints [33.344, -72.03, 117.725, 42.596, -54.303, -28.213] to (-191.86, -198.42, -8.35) mm, rotated rx -180 ry 0 rz -179 deg; joints [33.166, -73.039, 119.115, 42.219, -54.501, -27.785]
  MoveL 1285 to (-293.46, -198.42, -8.35) mm, rotated rx -180 ry 0 rz -179 deg; joints [35.779, -77.985, 125.639, 44.277, -56.874, -28.052]
  MoveC 1286 to (-306.16, -211.12, -8.35) mm, rotated rx 180 ry 0 rz -179 deg; joints [36.635, -78.166, 125.868, 45.153, -57.314, -28.499] to (-318.86, -198.42, -8.35) mm, rotated rx -180 ry 0 rz -179 deg; joints [36.491, -79.221, 127.19, 44.882, -57.434, -28.194]
  MoveL 1287 to (-395.06, -198.42, -8.35) mm, rotated rx -180 ry 0 rz -179 deg; joints [38.787, -82.934, 131.652, 46.921, -59.051, -28.81]
  MoveL 1288 to (-420.46, -198.42, -8.35) mm, rotated rx -180 ry 0 rz -179 deg; joints [39.609, -84.175, 133.076, 47.678, -59.573, -29.081]
  MoveC 1289 to (-433.16, -211.12, -8.35) mm, rotated rx -180 ry 0 rz -179 deg; joints [40.554, -84.291, 133.207, 48.625, -60.045, -29.547] to (-445.86, -198.42, -8.35) mm, rotated rx -180 ry 0 rz -179 deg; joints [40.462, -85.419, 134.468, 48.475, -60.088, -29.386]
  MoveL 1290 to (-471.26, -198.42, -8.35) mm, rotated rx -180 ry 0 rz -179 deg; joints [41.347, -86.666, 135.827, 49.312, -60.599, -29.726]
  MoveL 1291 to (-471.26, -350.82, -8.35) mm, rotated rx -180 ry 0 rz -179 deg; joints [47.144, -80.168, 128.356, 55.334, -63.035, -33.253]
  MoveL 1292 to (-14.06, -350.82, -8.35) mm, rotated rx -180 ry 0 rz -179 deg; joints [34.476, -59.692, 99.282, 47.136, -50.559, -34.392]
  MoveL 1293 to (-14.06, -198.42, -8.35) mm, rotated rx -180 ry 0 rz -179 deg; joints [29.357, -64.236, 106.363, 39.982, -49.728, -28.46]
  MoveC 1294 to (-13.87, -197.97, -8.35) mm, rotated rx 180 ry 0 rz -179 deg; joints [29.338, -64.238, 106.367, 39.959, -49.72, -28.444] to (-13.42, -197.78, -8.35) mm, rotated rx -180 ry 0 rz -179 deg; joints [29.323, -64.221, 106.34, 39.946, -49.706, -28.441]
  MoveL 1295 to (-12.79, -197.78, -8.35) mm, rotated rx 180 ry 0 rz -179 deg; joints [29.31, -64.189, 106.291, 39.941, -49.687, -28.446]
  MoveC 1296 to (-12.34, -197.78, -8.16) mm, rotated rx 180 ry 0 rz -179 deg; joints [29.302, -64.173, 106.252, 39.944, -49.665, -28.459] to (-12.15, -197.78, -7.72) mm, rotated rx -180 ry 0 rz -179 deg; joints [29.298, -64.179, 106.226, 39.958, -49.638, -28.484]
  Set speed (500.0 mm/s)
  MoveL 1297 to (-12.15, -197.78, 6) mm, rotated rx -180 ry 0 rz -179 deg; joints [29.298, -64.666, 105.857, 40.433, -48.984, -29.213]
  MoveL 1298 to (12.15, -197.78, 6) mm, rotated rx -180 ry 0 rz -179 deg; joints [28.842, -63.421, 103.963, 40.273, -48.267, -29.422]
  Set speed (25.4 mm/s)
  MoveL 1299 to (12.15, -197.78, -4.36) mm, rotated rx -180 ry 0 rz -179 deg; joints [28.842, -63.062, 104.242, 39.909, -48.756, -28.873]
  MoveC 1300 to (12.34, -197.78, -4.81) mm, rotated rx 180 ry 0 rz -179 deg; joints [28.839, -63.036, 104.24, 39.893, -48.771, -28.851] to (12.79, -197.79, -5) mm, rotated rx -180 ry 0 rz -179 deg; joints [28.831, -63.007, 104.209, 39.884, -48.766, -28.846]
  Set speed (50.8 mm/s)
  MoveL 1301 to (13.42, -197.79, -5) mm, rotated rx -180 ry 0 rz -179 deg; joints [28.819, -62.975, 104.159, 39.88, -48.747, -28.852]
  MoveC 1302 to (13.87, -197.97, -5) mm, rotated rx 180 ry 0 rz -179 deg; joints [28.817, -62.947, 104.116, 39.886, -48.735, -28.863] to (14.06, -198.42, -5) mm, rotated rx 180 ry 0 rz -179 deg; joints [28.829, -62.925, 104.083, 39.907, -48.732, -28.883]
  MoveL 1303 to (14.06, -350.82, -5) mm, rotated rx -180 ry 0 rz -179 deg; joints [33.894, -58.415, 96.973, 47.145, -49.527, -34.977]
  MoveL 1304 to (471.26, -350.82, -5) mm, rotated rx 180 ry 0 rz -179 deg; joints [26.49, -28.4, 43.798, 61.951, -30.357, -58.306]
  MoveL 1305 to (471.26, -198.42, -5) mm, rotated rx -180 ry 0 rz -179 deg; joints [22.262, -34.723, 55.676, 48.861, -30.201, -44.694]
  MoveL 1306 to (445.86, -198.42, -5) mm, rotated rx 180 ry 0 rz -179 deg; joints [22.549, -36.836, 59.576, 47.047, -31.596, -42.456]
  MoveC 1307 to (433.16, -211.12, -5) mm, rotated rx -180 ry 0 rz -179 deg; joints [23.063, -37.442, 60.688, 47.17, -32.287, -42.364] to (420.46, -198.42, -5) mm, rotated rx -180 ry 0 rz -179 deg; joints [22.843, -38.816, 63.199, 45.578, -32.925, -40.579]
  MoveL 1308 to (395.06, -198.42, -5) mm, rotated rx 180 ry 0 rz -179 deg; joints [23.144, -40.69, 66.596, 44.374, -34.196, -38.981]
  MoveL 1309 to (318.86, -198.42, -5) mm, rotated rx -180 ry 0 rz -179 deg; joints [24.098, -45.843, 75.773, 41.875, -37.711, -35.344]
  MoveC 1310 to (306.16, -211.12, -5) mm, rotated rx 180 ry 0 rz -179 deg; joints [24.654, -46.301, 76.577, 42.314, -38.29, -35.547] to (293.46, -198.42, -5) mm, rotated rx -180 ry 0 rz -179 deg; joints [24.434, -47.442, 78.568, 41.312, -38.798, -34.411]
  MoveL 1311 to (191.86, -198.42, -5) mm, rotated rx -180 ry 0 rz -179 deg; joints [25.873, -53.43, 88.792, 39.963, -42.796, -31.588]
  MoveC 1312 to (179.16, -211.12, -5) mm, rotated rx -180 ry 0 rz -179 deg; joints [26.475, -53.808, 89.423, 40.539, -43.307, -31.897] to (166.46, -198.42, -5) mm, rotated rx -180 ry 0 rz -179 deg; joints [26.258, -54.848, 91.152, 39.802, -43.72, -31.057]
  MoveL 1313 to (90.26, -198.42, -5) mm, rotated rx -180 ry 0 rz -179 deg; joints [27.486, -58.965, 97.857, 39.647, -46.332, -29.776]
  MoveL 1314 to (64.86, -198.42, -5) mm, rotated rx -180 ry 0 rz -179 deg; joints [27.92, -60.3, 99.981, 39.691, -47.154, -29.44]
  MoveC 1315 to (61.14, -207.4, -5) mm, rotated rx 180 ry 0 rz -179 deg; joints [28.292, -60.254, 99.909, 40.146, -47.317, -29.762] to (52.16, -211.12, -5) mm, rotated rx 180 ry 0 rz -179 deg; joints [28.577, -60.621, 100.487, 40.357, -47.621, -29.803]
  MoveL 1316 to (52.16, -211.12, -5) mm, rotated rx -180 ry 0 rz -179 deg; joints [28.577, -60.621, 100.487, 40.357, -47.621, -29.803]
  MoveC 1317 to (43.18, -207.4, -5) mm, rotated rx -180 ry 0 rz -179 deg; joints [28.611, -61.186, 101.376, 40.206, -47.885, -29.546] to (39.46, -198.42, -5) mm, rotated rx -180 ry 0 rz -179 deg; joints [28.368, -61.619, 102.055, 39.778, -47.954, -29.143]
  MoveL 1318 to (14.06, -198.42, -5) mm, rotated rx -180 ry 0 rz -179 deg; joints [28.829, -62.925, 104.083, 39.907, -48.732, -28.883]
  MoveC 1319 to (13.61, -198.23, -5) mm, rotated rx -180 ry 0 rz -179 deg; joints [28.831, -62.953, 104.126, 39.901, -48.744, -28.871] to (13.42, -197.79, -5) mm, rotated rx -180 ry 0 rz -179 deg; joints [28.819, -62.975, 104.159, 39.88, -48.747, -28.852]
  MoveL 1320 to (13.42, -197.15, -5) mm, rotated rx -180 ry 0 rz -179 deg; joints [28.797, -62.992, 104.186, 39.849, -48.744, -28.827]
  MoveC 1321 to (13.42, -196.7, -4.81) mm, rotated rx 180 ry 0 rz -179 deg; joints [28.781, -63.01, 104.199, 39.833, -48.732, -28.819] to (13.42, -196.52, -4.37) mm, rotated rx 180 ry 0 rz -179 deg; joints [28.775, -63.031, 104.195, 39.84, -48.71, -28.835]
  Set speed (500.0 mm/s)
  MoveL 1322 to (13.42, -196.51, 5) mm, rotated rx 180 ry 0 rz -179 deg; joints [28.775, -63.355, 103.943, 40.168, -48.268, -29.33]
  MoveL 1323 to (12.15, -197.79, 5) mm, rotated rx -180 ry 0 rz -179 deg; joints [28.842, -63.386, 103.99, 40.237, -48.314, -29.369]
  Set speed (25.4 mm/s)
  MoveL 1324 to (12.15, -197.78, 1) mm, rotated rx -180 ry 0 rz -179 deg; joints [28.842, -63.248, 104.099, 40.096, -48.503, -29.156]
  MoveL 1325 to (12.15, -197.78, -7.72) mm, rotated rx 180 ry 0 rz -179 deg; joints [28.842, -62.944, 104.331, 39.794, -48.914, -28.698]
  MoveC 1326 to (12.34, -197.78, -8.16) mm, rotated rx -180 ry 0 rz -179 deg; joints [28.839, -62.919, 104.328, 39.777, -48.929, -28.676] to (12.79, -197.79, -8.35) mm, rotated rx -180 ry 0 rz -179 deg; joints [28.831, -62.889, 104.297, 39.768, -48.925, -28.671]
  Set speed (50.8 mm/s)
  MoveL 1327 to (13.42, -197.78, -8.35) mm, rotated rx -180 ry 0 rz -179 deg; joints [28.819, -62.857, 104.247, 39.765, -48.905, -28.677]
  MoveC 1328 to (13.87, -197.97, -8.35) mm, rotated rx 180 ry 0 rz -179 deg; joints [28.817, -62.829, 104.204, 39.771, -48.893, -28.688] to (14.06, -198.42, -8.35) mm, rotated rx -180 ry 0 rz -179 deg; joints [28.829, -62.808, 104.171, 39.792, -48.89, -28.708]
  MoveL 1329 to (14.06, -350.82, -8.35) mm, rotated rx 180 ry 0 rz -179 deg; joints [33.894, -58.306, 97.061, 47.022, -49.66, -34.788]
  MoveL 1330 to (471.26, -350.82, -8.35) mm, rotated rx -180 ry 0 rz -179 deg; joints [26.49, -28.362, 43.956, 61.656, -30.45, -57.964]
  MoveL 1331 to (471.26, -198.42, -8.35) mm, rotated rx 180 ry 0 rz -179 deg; joints [22.262, -34.663, 55.799, 48.625, -30.322, -44.421]
  MoveL 1332 to (445.86, -198.42, -8.35) mm, rotated rx 180 ry 0 rz -179 deg; joints [22.549, -36.77, 59.692, 46.832, -31.72, -42.203]
  MoveC 1333 to (433.16, -211.12, -8.35) mm, rotated rx 180 ry 0 rz -179 deg; joints [23.063, -37.374, 60.801, 46.961, -32.41, -42.117] to (420.46, -198.42, -8.35) mm, rotated rx -180 ry 0 rz -179 deg; joints [22.843, -38.746, 63.309, 45.38, -33.052, -40.343]
  MoveL 1334 to (395.06, -198.42, -8.35) mm, rotated rx 180 ry 0 rz -179 deg; joints [23.144, -40.616, 66.702, 44.19, -34.325, -38.758]
  MoveL 1335 to (318.86, -198.42, -8.35) mm, rotated rx 180 ry 0 rz -179 deg; joints [24.098, -45.759, 75.87, 41.719, -37.846, -35.147]
  MoveC 1336 to (306.16, -211.12, -8.35) mm, rotated rx -180 ry 0 rz -179 deg; joints [24.654, -46.216, 76.673, 42.16, -38.424, -35.351] to (293.46, -198.42, -8.35) mm, rotated rx -180 ry 0 rz -179 deg; joints [24.434, -47.354, 78.663, 41.163, -38.935, -34.219]
  MoveL 1337 to (191.86, -198.42, -8.35) mm, rotated rx 180 ry 0 rz -179 deg; joints [25.873, -53.331, 88.882, 39.833, -42.941, -31.41]
  MoveC 1338 to (179.16, -211.12, -8.35) mm, rotated rx -180 ry 0 rz -179 deg; joints [26.475, -53.708, 89.512, 40.409, -43.45, -31.718] to (166.46, -198.42, -8.35) mm, rotated rx -180 ry 0 rz -179 deg; joints [26.258, -54.747, 91.241, 39.675, -43.866, -30.881]
  MoveL 1339 to (90.26, -198.42, -8.35) mm, rotated rx 180 ry 0 rz -179 deg; joints [27.486, -58.856, 97.945, 39.527, -46.484, -29.603]
  MoveL 1340 to (64.86, -198.42, -8.35) mm, rotated rx -180 ry 0 rz -179 deg; joints [27.92, -60.188, 100.069, 39.573, -47.308, -29.266]
  MoveC 1341 to (61.14, -207.4, -8.35) mm, rotated rx -180 ry 0 rz -179 deg; joints [28.292, -60.142, 99.997, 40.028, -47.47, -29.587] to (52.16, -211.12, -8.35) mm, rotated rx 180 ry 0 rz -179 deg; joints [28.577, -60.508, 100.575, 40.239, -47.774, -29.627]
  MoveL 1342 to (52.16, -211.12, -8.35) mm, rotated rx 180 ry 0 rz -179 deg; joints [28.577, -60.508, 100.575, 40.239, -47.774, -29.627]
  MoveC 1343 to (43.18, -207.4, -8.35) mm, rotated rx 180 ry 0 rz -179 deg; joints [28.611, -61.072, 101.465, 40.088, -48.039, -29.371] to (39.46, -198.42, -8.35) mm, rotated rx 180 ry 0 rz -179 deg; joints [28.368, -61.505, 102.143, 39.662, -48.11, -28.968]
  MoveL 1344 to (14.06, -198.42, -8.35) mm, rotated rx -180 ry 0 rz -179 deg; joints [28.829, -62.808, 104.171, 39.792, -48.89, -28.708]
  MoveC 1345 to (13.61, -198.23, -8.35) mm, rotated rx -180 ry 0 rz -179 deg; joints [28.831, -62.835, 104.214, 39.785, -48.902, -28.696] to (13.42, -197.79, -8.35) mm, rotated rx -180 ry 0 rz -179 deg; joints [28.819, -62.857, 104.247, 39.765, -48.905, -28.677]
  MoveL 1346 to (13.42, -197.15, -8.35) mm, rotated rx -180 ry 0 rz -179 deg; joints [28.797, -62.874, 104.274, 39.734, -48.902, -28.652]
  MoveC 1347 to (13.42, -196.7, -8.16) mm, rotated rx -180 ry 0 rz -179 deg; joints [28.781, -62.893, 104.288, 39.718, -48.891, -28.644] to (13.42, -196.52, -7.72) mm, rotated rx -180 ry 0 rz -179 deg; joints [28.775, -62.914, 104.284, 39.724, -48.868, -28.66]
  Set speed (500.0 mm/s)
  MoveL 1348 to (13.42, -196.51, 6) mm, rotated rx -180 ry 0 rz -179 deg; joints [28.775, -63.39, 103.916, 40.203, -48.221, -29.383]
  MoveL 1349 to (12.15, -384.12, 6) mm, rotated rx -180 ry 0 rz -179 deg; joints [34.97, -57.762, 95.065, 49.092, -49.321, -36.953]
  Set speed (25.4 mm/s)
  MoveL 1350 to (12.15, -384.12, -4.36) mm, rotated rx -180 ry 0 rz -179 deg; joints [34.97, -57.437, 95.345, 48.703, -49.718, -36.355]
  MoveC 1351 to (12.34, -384.12, -4.81) mm, rotated rx -180 ry 0 rz -179 deg; joints [34.966, -57.414, 95.342, 48.686, -49.729, -36.332] to (12.79, -384.12, -5) mm, rotated rx -180 ry 0 rz -179 deg; joints [34.957, -57.386, 95.311, 48.679, -49.722, -36.328]
  Set speed (50.8 mm/s)
  MoveL 1352 to (13.42, -384.12, -5) mm, rotated rx -180 ry 0 rz -179 deg; joints [34.944, -57.354, 95.26, 48.677, -49.701, -36.339]
  MoveC 1353 to (13.87, -384.31, -5) mm, rotated rx 180 ry 0 rz -179 deg; joints [34.94, -57.326, 95.213, 48.685, -49.687, -36.354] to (14.06, -384.76, -5) mm, rotated rx -180 ry 0 rz -179 deg; joints [34.95, -57.301, 95.174, 48.705, -49.683, -36.376]
  MoveL 1354 to (14.06, -537.16, -5) mm, rotated rx -180 ry 0 rz -179 deg; joints [39.383, -51.773, 86.002, 55.58, -50.28, -43.003]
  MoveL 1355 to (471.26, -537.16, -5) mm, rotated rx 180 ry 0 rz 151 deg; joints [26.498, -21.395, 30.303, -21.566, -9.566, 21.293]
  MoveL 1356 to (471.26, -384.76, -5) mm, rotated rx -180 ry 0 rz -179 deg; joints [27.394, -26.516, 40.202, 65.46, -30.384, -62.109]
  MoveL 1357 to (445.86, -384.76, -5) mm, rotated rx 180 ry 0 rz -179 deg; joints [27.731, -29.329, 45.561, 61.999, -31.804, -57.967]
  MoveC 1358 to (433.16, -397.46, -5) mm, rotated rx -180 ry 0 rz -179 deg; joints [28.241, -29.96, 46.755, 61.721, -32.501, -57.467] to (420.46, -384.76, -5) mm, rotated rx -180 ry 0 rz -179 deg; joints [28.076, -31.796, 50.215, 59.36, -33.162, -54.717]
  MoveL 1359 to (395.06, -384.76, -5) mm, rotated rx -180 ry 0 rz -179 deg; joints [28.43, -34.029, 54.387, 57.275, -34.465, -52.067]
  MoveL 1360 to (318.86, -384.76, -5) mm, rotated rx -180 ry 0 rz -179 deg; joints [29.543, -39.833, 65.046, 53.071, -38.084, -46.321]
  MoveC 1361 to (306.16, -397.46, -5) mm, rotated rx -180 ry 0 rz -179 deg; joints [30.091, -40.229, 65.762, 53.356, -38.673, -46.385] to (293.46, -384.76, -5) mm, rotated rx -180 ry 0 rz -179 deg; joints [29.933, -41.563, 68.168, 52.125, -39.209, -44.892]
  MoveL 1362 to (191.86, -384.76, -5) mm, rotated rx -180 ry 0 rz -179 deg; joints [31.594, -47.839, 79.258, 49.717, -43.373, -40.617]
  MoveC 1363 to (179.16, -397.46, -5) mm, rotated rx -180 ry 0 rz -179 deg; joints [32.183, -48.132, 79.766, 50.191, -43.896, -40.847] to (166.46, -384.76, -5) mm, rotated rx -180 ry 0 rz -179 deg; joints [32.036, -49.286, 81.759, 49.37, -44.343, -39.812]
  MoveL 1364 to (90.26, -384.76, -5) mm, rotated rx 180 ry 0 rz -179 deg; joints [33.435, -53.418, 88.771, 48.77, -47.107, -37.835]
  MoveL 1365 to (64.86, -384.76, -5) mm, rotated rx -180 ry 0 rz -179 deg; joints [33.926, -54.737, 90.967, 48.695, -47.985, -37.298]
  MoveC 1366 to (61.14, -393.74, -5) mm, rotated rx -180 ry 0 rz -179 deg; joints [34.271, -54.627, 90.785, 49.112, -48.148, -37.617] to (52.16, -397.46, -5) mm, rotated rx -180 ry 0 rz -179 deg; joints [34.562, -54.961, 91.337, 49.273, -48.468, -37.6]
  MoveL 1367 to (52.16, -397.46, -5) mm, rotated rx -180 ry 0 rz -179 deg; joints [34.562, -54.961, 91.337, 49.273, -48.468, -37.6]
  MoveC 1368 to (43.18, -393.74, -5) mm, rotated rx -180 ry 0 rz -179 deg; joints [34.63, -55.542, 92.297, 49.092, -48.756, -37.266] to (39.46, -384.76, -5) mm, rotated rx -180 ry 0 rz -179 deg; joints [34.431, -56.03, 93.1, 48.675, -48.844, -36.813]
  MoveL 1369 to (14.06, -384.76, -5) mm, rotated rx -180 ry 0 rz -179 deg; joints [34.95, -57.301, 95.174, 48.705, -49.683, -36.376]
  MoveC 1370 to (13.61, -384.57, -5) mm, rotated rx -180 ry 0 rz -179 deg; joints [34.954, -57.33, 95.22, 48.697, -49.697, -36.36] to (13.42, -384.12, -5) mm, rotated rx 180 ry 0 rz -179 deg; joints [34.944, -57.354, 95.26, 48.677, -49.701, -36.339]
  MoveL 1371 to (13.42, -383.49, -5) mm, rotated rx -180 ry 0 rz -179 deg; joints [34.924, -57.375, 95.294, 48.648, -49.698, -36.312]
  MoveC 1372 to (13.42, -383.04, -4.81) mm, rotated rx 180 ry 0 rz -179 deg; joints [34.91, -57.396, 95.313, 48.634, -49.689, -36.304] to (13.42, -382.85, -4.37) mm, rotated rx 180 ry 0 rz -179 deg; joints [34.905, -57.417, 95.311, 48.643, -49.671, -36.322]
  Set speed (500.0 mm/s)
  MoveL 1373 to (13.42, -382.85, 5) mm, rotated rx -180 ry 0 rz -179 deg; joints [34.905, -57.71, 95.059, 48.993, -49.312, -36.863]
  MoveL 1374 to (12.15, -384.12, 5) mm, rotated rx -180 ry 0 rz -179 deg; joints [34.97, -57.731, 95.093, 49.054, -49.359, -36.895]
  Set speed (25.4 mm/s)
  MoveL 1375 to (12.15, -384.12, 1) mm, rotated rx -180 ry 0 rz -179 deg; joints [34.97, -57.606, 95.201, 48.903, -49.512, -36.663]
  MoveL 1376 to (12.15, -384.12, -7.72) mm, rotated rx 180 ry 0 rz -179 deg; joints [34.97, -57.331, 95.433, 48.58, -49.847, -36.163]
  MoveC 1377 to (12.34, -384.12, -8.16) mm, rotated rx -180 ry 0 rz -179 deg; joints [34.966, -57.307, 95.43, 48.563, -49.858, -36.141] to (12.79, -384.12, -8.35) mm, rotated rx -180 ry 0 rz -179 deg; joints [34.957, -57.279, 95.399, 48.555, -49.851, -36.137]
  Set speed (50.8 mm/s)
  MoveL 1378 to (13.42, -384.12, -8.35) mm, rotated rx 180 ry 0 rz -179 deg; joints [34.944, -57.248, 95.348, 48.554, -49.83, -36.148]
  MoveC 1379 to (13.87, -384.31, -8.35) mm, rotated rx -180 ry 0 rz -179 deg; joints [34.94, -57.219, 95.302, 48.561, -49.816, -36.163] to (14.06, -384.76, -8.35) mm, rotated rx -180 ry 0 rz -179 deg; joints [34.95, -57.195, 95.262, 48.581, -49.812, -36.184]
  MoveL 1380 to (14.06, -537.16, -8.35) mm, rotated rx 180 ry 0 rz -179 deg; joints [39.383, -51.677, 86.093, 55.453, -50.385, -42.803]
  MoveL 1381 to (471.26, -537.16, -8.35) mm, rotated rx 180 ry 0 rz 151 deg; joints [26.498, -21.406, 30.555, -21.051, -9.791, 20.771]
  MoveL 1382 to (471.26, -384.76, -8.35) mm, rotated rx -180 ry 0 rz -179 deg; joints [27.394, -26.487, 40.377, 65.144, -30.469, -61.743]
  MoveL 1383 to (445.86, -384.76, -8.35) mm, rotated rx -180 ry 0 rz -179 deg; joints [27.731, -29.286, 45.712, 61.724, -31.895, -57.643]
  MoveC 1384 to (433.16, -397.46, -8.35) mm, rotated rx -180 ry 0 rz -179 deg; joints [28.241, -29.915, 46.902, 61.457, -32.592, -57.154] to (420.46, -384.76, -8.35) mm, rotated rx -180 ry 0 rz -179 deg; joints [28.076, -31.745, 50.352, 59.113, -33.258, -54.422]
  MoveL 1385 to (395.06, -384.76, -8.35) mm, rotated rx -180 ry 0 rz -179 deg; joints [28.43, -33.971, 54.513, 57.05, -34.565, -51.793]
  MoveL 1386 to (318.86, -384.76, -8.35) mm, rotated rx 180 ry 0 rz -179 deg; joints [29.543, -39.761, 65.154, 52.888, -38.193, -46.089]
  MoveC 1387 to (306.16, -397.46, -8.35) mm, rotated rx 180 ry 0 rz -179 deg; joints [30.091, -40.155, 65.869, 53.176, -38.78, -46.155] to (293.46, -384.76, -8.35) mm, rotated rx -180 ry 0 rz -179 deg; joints [29.933, -41.487, 68.272, 51.951, -39.319, -44.668]
  MoveL 1388 to (191.86, -384.76, -8.35) mm, rotated rx -180 ry 0 rz -179 deg; joints [31.594, -47.75, 79.352, 49.57, -43.491, -40.415]
  MoveC 1389 to (179.16, -397.46, -8.35) mm, rotated rx 180 ry 0 rz -179 deg; joints [32.183, -48.043, 79.86, 50.045, -44.014, -40.645] to (166.46, -384.76, -8.35) mm, rotated rx -180 ry 0 rz -179 deg; joints [32.036, -49.195, 81.852, 49.227, -44.463, -39.612]
  MoveL 1390 to (90.26, -384.76, -8.35) mm, rotated rx 180 ry 0 rz -179 deg; joints [33.435, -53.319, 88.861, 48.639, -47.232, -37.642]
  MoveL 1391 to (64.86, -384.76, -8.35) mm, rotated rx 180 ry 0 rz -179 deg; joints [33.926, -54.635, 91.056, 48.567, -48.111, -37.106]
  MoveC 1392 to (61.14, -393.74, -8.35) mm, rotated rx -180 ry 0 rz -179 deg; joints [34.271, -54.526, 90.874, 48.983, -48.272, -37.424] to (52.16, -397.46, -8.35) mm, rotated rx -180 ry 0 rz -179 deg; joints [34.562, -54.859, 91.426, 49.145, -48.592, -37.407]
  MoveL 1393 to (52.16, -397.46, -8.35) mm, rotated rx -180 ry 0 rz -179 deg; joints [34.562, -54.859, 91.426, 49.145, -48.592, -37.407]
  MoveC 1394 to (43.18, -393.74, -8.35) mm, rotated rx 180 ry 0 rz -179 deg; joints [34.63, -55.439, 92.385, 48.966, -48.882, -37.074] to (39.46, -384.76, -8.35) mm, rotated rx -180 ry 0 rz -179 deg; joints [34.431, -55.927, 93.188, 48.549, -48.971, -36.622]
  MoveL 1395 to (14.06, -384.76, -8.35) mm, rotated rx -180 ry 0 rz -179 deg; joints [34.95, -57.195, 95.262, 48.581, -49.812, -36.184]
  MoveC 1396 to (13.61, -384.57, -8.35) mm, rotated rx -180 ry 0 rz -179 deg; joints [34.954, -57.224, 95.309, 48.574, -49.826, -36.169] to (13.42, -384.12, -8.35) mm, rotated rx 180 ry 0 rz -179 deg; joints [34.944, -57.248, 95.348, 48.554, -49.83, -36.148]
  MoveL 1397 to (13.42, -383.49, -8.35) mm, rotated rx -180 ry 0 rz -179 deg; joints [34.924, -57.269, 95.382, 48.525, -49.827, -36.121]
  MoveC 1398 to (13.42, -383.04, -8.16) mm, rotated rx -180 ry 0 rz -179 deg; joints [34.91, -57.29, 95.402, 48.511, -49.818, -36.113] to (13.42, -382.85, -7.72) mm, rotated rx 180 ry 0 rz -179 deg; joints [34.905, -57.31, 95.4, 48.519, -49.8, -36.131]
  Set speed (500.0 mm/s)
  MoveL 1399 to (13.42, -382.85, 6) mm, rotated rx -180 ry 0 rz -179 deg; joints [34.905, -57.741, 95.032, 49.031, -49.273, -36.921]
  MoveL 1400 to (-13.42, -382.85, 6) mm, rotated rx 180 ry 0 rz -179 deg; joints [35.469, -59.07, 97.163, 49.11, -50.136, -36.509]
  Set speed (25.4 mm/s)
  MoveL 1401 to (-13.42, -382.85, -4.36) mm, rotated rx 180 ry 0 rz -179 deg; joints [35.469, -58.737, 97.442, 48.728, -50.538, -35.911]
  MoveC 1402 to (-13.42, -383.04, -4.81) mm, rotated rx -180 ry 0 rz -179 deg; joints [35.474, -58.717, 97.444, 48.72, -50.556, -35.892] to (-13.42, -383.49, -5) mm, rotated rx 180 ry 0 rz -179 deg; joints [35.488, -58.696, 97.424, 48.733, -50.565, -35.9]
  Set speed (50.8 mm/s)
  MoveL 1403 to (-13.42, -384.12, -5) mm, rotated rx 180 ry 0 rz -179 deg; joints [35.508, -58.674, 97.39, 48.762, -50.568, -35.926]
  MoveC 1404 to (-13.61, -384.57, -5) mm, rotated rx -180 ry 0 rz -179 deg; joints [35.526, -58.668, 97.381, 48.783, -50.577, -35.941] to (-14.06, -384.76, -5) mm, rotated rx -180 ry 0 rz -179 deg; joints [35.541, -58.684, 97.406, 48.793, -50.592, -35.942]
  MoveL 1405 to (-39.46, -384.76, -5) mm, rotated rx -180 ry 0 rz -179 deg; joints [36.091, -59.913, 99.368, 48.92, -51.395, -35.593]
  MoveC 1406 to (-52.16, -397.46, -5) mm, rotated rx 180 ry 0 rz -179 deg; joints [36.767, -60.088, 99.646, 49.559, -51.858, -35.928] to (-64.86, -384.76, -5) mm, rotated rx -180 ry 0 rz -179 deg; joints [36.656, -61.125, 101.281, 49.089, -52.183, -35.282]
  MoveL 1407 to (-90.26, -384.76, -5) mm, rotated rx -180 ry 0 rz -179 deg; joints [37.237, -62.321, 103.147, 49.299, -52.956, -35.006]
  MoveL 1408 to (-166.46, -384.76, -5) mm, rotated rx -180 ry 0 rz -179 deg; joints [39.081, -65.822, 108.485, 50.157, -55.193, -34.374]
  MoveC 1409 to (-179.16, -397.46, -5) mm, rotated rx -180 ry 0 rz -179 deg; joints [39.812, -65.939, 108.661, 50.857, -55.645, -34.735] to (-191.86, -384.76, -5) mm, rotated rx -180 ry 0 rz -179 deg; joints [39.732, -66.963, 110.182, 50.515, -55.914, -34.224]
  MoveL 1410 to (-293.46, -384.76, -5) mm, rotated rx 180 ry 0 rz -179 deg; joints [42.531, -71.418, 116.59, 52.291, -58.7, -33.899]
  MoveC 1411 to (-306.16, -397.46, -5) mm, rotated rx -180 ry 0 rz -179 deg; joints [43.321, -71.474, 116.667, 53.044, -59.156, -34.273] to (-318.86, -384.76, -5) mm, rotated rx -180 ry 0 rz -179 deg; joints [43.283, -72.507, 118.1, 52.818, -59.376, -33.883]
  MoveL 1412 to (-395.06, -384.76, -5) mm, rotated rx 180 ry 0 rz -179 deg; joints [45.677, -75.717, 122.42, 54.594, -61.37, -33.983]
  MoveL 1413 to (-420.46, -384.76, -5) mm, rotated rx -180 ry 0 rz -179 deg; joints [46.523, -76.768, 123.791, 55.25, -62.027, -34.064]
  MoveC 1414 to (-433.16, -397.46, -5) mm, rotated rx -180 ry 0 rz -179 deg; joints [47.373, -76.751, 123.768, 56.046, -62.502, -34.439] to (-445.86, -384.76, -5) mm, rotated rx -180 ry 0 rz -179 deg; joints [47.394, -77.81, 125.127, 55.937, -62.681, -34.169]
  MoveL 1415 to (-471.26, -384.76, -5) mm, rotated rx -180 ry 0 rz -179 deg; joints [48.291, -78.843, 126.428, 56.656, -63.335, -34.296]
  MoveL 1416 to (-471.26, -537.16, -5) mm, rotated rx -180 ry 0 rz -179 deg; joints [52.884, -72.054, 117.474, 61.676, -64.942, -38.16]
  MoveL 1417 to (-14.06, -537.16, -5) mm, rotated rx 180 ry 0 rz -179 deg; joints [40.003, -53.151, 88.324, 55.533, -51.234, -42.37]
  MoveL 1418 to (-14.06, -384.76, -5) mm, rotated rx -180 ry 0 rz -179 deg; joints [35.541, -58.684, 97.406, 48.793, -50.592, -35.942]
  MoveC 1419 to (-13.87, -384.31, -5) mm, rotated rx -180 ry 0 rz -179 deg; joints [35.523, -58.69, 97.415, 48.772, -50.584, -35.927] to (-13.42, -384.12, -5) mm, rotated rx 180 ry 0 rz -179 deg; joints [35.508, -58.674, 97.39, 48.762, -50.568, -35.926]
  MoveL 1420 to (-12.79, -384.12, -5) mm, rotated rx 180 ry 0 rz -179 deg; joints [35.494, -58.643, 97.341, 48.759, -50.548, -35.935]
  MoveC 1421 to (-12.34, -384.12, -4.81) mm, rotated rx 180 ry 0 rz -179 deg; joints [35.485, -58.627, 97.3, 48.764, -50.527, -35.952] to (-12.15, -384.12, -4.37) mm, rotated rx -180 ry 0 rz -179 deg; joints [35.481, -58.633, 97.274, 48.78, -50.503, -35.981]
  Set speed (500.0 mm/s)
  MoveL 1422 to (-12.15, -384.12, 5) mm, rotated rx -180 ry 0 rz -179 deg; joints [35.481, -58.933, 97.022, 49.125, -50.141, -36.521]
  MoveL 1423 to (-13.42, -382.85, 5) mm, rotated rx -180 ry 0 rz -179 deg; joints [35.469, -59.038, 97.19, 49.073, -50.175, -36.451]
  Set speed (25.4 mm/s)
  MoveL 1424 to (-13.42, -382.85, 1) mm, rotated rx 180 ry 0 rz -179 deg; joints [35.469, -58.91, 97.298, 48.924, -50.33, -36.219]
  MoveL 1425 to (-13.42, -382.85, -7.72) mm, rotated rx 180 ry 0 rz -179 deg; joints [35.469, -58.629, 97.53, 48.606, -50.668, -35.719]
  MoveC 1426 to (-13.42, -383.04, -8.16) mm, rotated rx 180 ry 0 rz -179 deg; joints [35.474, -58.608, 97.532, 48.598, -50.686, -35.701] to (-13.42, -383.49, -8.35) mm, rotated rx 180 ry 0 rz -179 deg; joints [35.488, -58.587, 97.513, 48.612, -50.696, -35.709]
  Set speed (50.8 mm/s)
  MoveL 1427 to (-13.42, -384.12, -8.35) mm, rotated rx -180 ry 0 rz -179 deg; joints [35.508, -58.565, 97.478, 48.641, -50.698, -35.734]
  MoveC 1428 to (-13.61, -384.57, -8.35) mm, rotated rx -180 ry 0 rz -179 deg; joints [35.526, -58.559, 97.469, 48.662, -50.707, -35.75] to (-14.06, -384.76, -8.35) mm, rotated rx -180 ry 0 rz -179 deg; joints [35.541, -58.575, 97.494, 48.672, -50.722, -35.751]
  MoveL 1429 to (-39.46, -384.76, -8.35) mm, rotated rx -180 ry 0 rz -179 deg; joints [36.091, -59.802, 99.456, 48.8, -51.526, -35.401]
  MoveC 1430 to (-52.16, -397.46, -8.35) mm, rotated rx -180 ry 0 rz -179 deg; joints [36.767, -59.977, 99.734, 49.44, -51.987, -35.736] to (-64.86, -384.76, -8.35) mm, rotated rx -180 ry 0 rz -179 deg; joints [36.656, -61.011, 101.369, 48.971, -52.315, -35.089]
  MoveL 1431 to (-90.26, -384.76, -8.35) mm, rotated rx -180 ry 0 rz -179 deg; joints [37.237, -62.204, 103.236, 49.182, -53.089, -34.812]
  MoveL 1432 to (-166.46, -384.76, -8.35) mm, rotated rx -180 ry 0 rz -179 deg; joints [39.081, -65.698, 108.574, 50.043, -55.329, -34.176]
  MoveC 1433 to (-179.16, -397.46, -8.35) mm, rotated rx -180 ry 0 rz -179 deg; joints [39.812, -65.816, 108.75, 50.744, -55.779, -34.535] to (-191.86, -384.76, -8.35) mm, rotated rx 180 ry 0 rz -179 deg; joints [39.732, -66.837, 110.272, 50.403, -56.052, -34.024]
  MoveL 1434 to (-293.46, -384.76, -8.35) mm, rotated rx -180 ry 0 rz -179 deg; joints [42.531, -71.282, 116.682, 52.182, -58.84, -33.689]
  MoveC 1435 to (-306.16, -397.46, -8.35) mm, rotated rx -180 ry 0 rz -179 deg; joints [43.321, -71.338, 116.759, 52.936, -59.294, -34.061] to (-318.86, -384.76, -8.35) mm, rotated rx -180 ry 0 rz -179 deg; joints [43.283, -72.368, 118.193, 52.71, -59.516, -33.669]
  MoveL 1436 to (-395.06, -384.76, -8.35) mm, rotated rx -180 ry 0 rz -179 deg; joints [45.677, -75.57, 122.516, 54.487, -61.51, -33.759]
  MoveL 1437 to (-420.46, -384.76, -8.35) mm, rotated rx -180 ry 0 rz -179 deg; joints [46.523, -76.619, 123.887, 55.143, -62.167, -33.836]
  MoveC 1438 to (-433.16, -397.46, -8.35) mm, rotated rx 180 ry 0 rz -179 deg; joints [47.373, -76.602, 123.864, 55.941, -62.639, -34.21] to (-445.86, -384.76, -8.35) mm, rotated rx -180 ry 0 rz -179 deg; joints [47.394, -77.659, 125.224, 55.831, -62.821, -33.937]
  MoveL 1439 to (-471.26, -384.76, -8.35) mm, rotated rx 180 ry 0 rz -179 deg; joints [48.291, -78.689, 126.526, 56.55, -63.474, -34.06]
  MoveL 1440 to (-471.26, -537.16, -8.35) mm, rotated rx -180 ry 0 rz -179 deg; joints [52.884, -71.916, 117.566, 61.581, -65.051, -37.937]
  MoveL 1441 to (-14.06, -537.16, -8.35) mm, rotated rx 180 ry 0 rz -179 deg; joints [40.003, -53.053, 88.414, 55.409, -51.34, -42.172]
  MoveL 1442 to (-14.06, -384.76, -8.35) mm, rotated rx 180 ry 0 rz -179 deg; joints [35.541, -58.575, 97.494, 48.672, -50.722, -35.751]
  MoveC 1443 to (-13.87, -384.31, -8.35) mm, rotated rx 180 ry 0 rz -179 deg; joints [35.523, -58.581, 97.504, 48.651, -50.714, -35.735] to (-13.42, -384.12, -8.35) mm, rotated rx -180 ry 0 rz -179 deg; joints [35.508, -58.565, 97.478, 48.641, -50.698, -35.734]
  MoveL 1444 to (-12.79, -384.12, -8.35) mm, rotated rx -180 ry 0 rz -179 deg; joints [35.494, -58.535, 97.429, 48.638, -50.678, -35.743]
  MoveC 1445 to (-12.34, -384.12, -8.16) mm, rotated rx -180 ry 0 rz -179 deg; joints [35.485, -58.519, 97.389, 48.643, -50.657, -35.761] to (-12.15, -384.12, -7.72) mm, rotated rx -180 ry 0 rz -179 deg; joints [35.481, -58.524, 97.362, 48.658, -50.633, -35.789]
  Set speed (500.0 mm/s)
  MoveL 1446 to (-12.15, -384.12, 6) mm, rotated rx -180 ry 0 rz -179 deg; joints [35.481, -58.965, 96.995, 49.162, -50.102, -36.579]
  MoveL 1447 to (-52.79, 196.52, 6) mm, rotated rx -180 ry 0 rz -179 deg; joints [14.058, -75.024, 120.57, 19.331, -47.206, -13.405]
  Set speed (25.4 mm/s)
  MoveL 1448 to (-52.79, 196.52, -4.36) mm, rotated rx 180 ry 0 rz -179 deg; joints [14.058, -74.586, 120.868, 19.109, -47.901, -13.076]
  MoveC 1449 to (-52.79, 196.7, -4.81) mm, rotated rx -180 ry 0 rz -179 deg; joints [14.05, -74.569, 120.884, 19.089, -47.93, -13.055] to (-52.79, 197.15, -5) mm, rotated rx -180 ry 0 rz -179 deg; joints [14.03, -74.567, 120.897, 19.058, -47.94, -13.03]
  Set speed (50.8 mm/s)
  MoveL 1450 to (-52.79, 197.78, -5) mm, rotated rx -180 ry 0 rz -179 deg; joints [14.001, -74.576, 120.908, 19.02, -47.936, -13.004]
  MoveC 1451 to (-52.61, 198.23, -5) mm, rotated rx -180 ry 0 rz -179 deg; joints [13.979, -74.571, 120.902, 18.991, -47.93, -12.985] to (-52.16, 198.42, -5) mm, rotated rx 180 ry 0 rz -179 deg; joints [13.966, -74.548, 120.871, 18.977, -47.919, -12.977]
  MoveL 1452 to (-14.06, 198.42, -5) mm, rotated rx 180 ry 0 rz -179 deg; joints [13.585, -72.397, 117.949, 18.701, -47.104, -12.975]
  MoveL 1453 to (-14.06, 350.82, -5) mm, rotated rx -180 ry 0 rz -179 deg; joints [6.808, -73.808, 119.875, 9.412, -46.456, -6.515]
  MoveL 1454 to (-39.46, 350.82, -5) mm, rotated rx -180 ry 0 rz -179 deg; joints [6.927, -75.276, 121.84, 9.498, -46.958, -6.515]
  MoveC 1455 to (-52.16, 338.12, -5) mm, rotated rx -180 ry 0 rz -179 deg; joints [7.58, -75.933, 122.705, 10.35, -47.24, -7.068] to (-64.86, 350.82, -5) mm, rotated rx -180 ry 0 rz -179 deg; joints [7.051, -76.756, 123.775, 9.596, -47.422, -6.526]
  MoveL 1456 to (-90.26, 350.82, -5) mm, rotated rx -180 ry 0 rz -179 deg; joints [7.181, -78.249, 125.682, 9.707, -47.844, -6.549]
  MoveL 1457 to (-166.46, 350.82, -5) mm, rotated rx -180 ry 0 rz -179 deg; joints [7.604, -82.831, 131.238, 10.122, -48.853, -6.699]
  MoveC 1458 to (-179.16, 338.12, -5) mm, rotated rx 180 ry 0 rz -179 deg; joints [8.339, -83.517, 132.03, 11.072, -49.047, -7.309] to (-191.86, 350.82, -5) mm, rotated rx -180 ry 0 rz -179 deg; joints [7.759, -84.402, 133.037, 10.29, -49.095, -6.779]
  MoveL 1459 to (-293.46, 350.82, -5) mm, rotated rx 180 ry 0 rz -179 deg; joints [8.456, -90.994, 139.976, 11.147, -49.521, -7.289]
  MoveC 1460 to (-306.16, 338.12, -5) mm, rotated rx -180 ry 0 rz -179 deg; joints [9.296, -91.74, 140.698, 12.244, -49.61, -8.005] to (-318.86, 350.82, -5) mm, rotated rx 180 ry 0 rz -179 deg; joints [8.653, -92.739, 141.645, 11.417, -49.473, -7.476]
  MoveL 1461 to (-395.06, 350.82, -5) mm, rotated rx 180 ry 0 rz -179 deg; joints [9.312, -98.276, 146.49, 12.403, -48.885, -8.229]
  MoveL 1462 to (-420.46, 350.82, -5) mm, rotated rx -180 ry 0 rz -179 deg; joints [9.558, -100.242, 148.046, 12.805, -48.521, -8.561]
  MoveC 1463 to (-433.16, 338.12, -5) mm, rotated rx -180 ry 0 rz -179 deg; joints [10.536, -101.089, 148.691, 14.136, -48.478, -9.478] to (-445.86, 350.82, -5) mm, rotated rx -180 ry 0 rz -179 deg; joints [9.818, -102.28, 149.571, 13.252, -48.062, -8.945]
  MoveL 1464 to (-471.26, 350.82, -5) mm, rotated rx -180 ry 0 rz -179 deg; joints [10.095, -104.395, 151.064, 13.753, -47.5, -9.389]
  MoveL 1465 to (-471.26, 198.42, -5) mm, rotated rx -180 ry 0 rz -179 deg; joints [20.36, -101.255, 148.815, 26.695, -50.754, -17.647]
  MoveL 1466 to (-445.86, 198.42, -5) mm, rotated rx -180 ry 0 rz -179 deg; joints [19.804, -99.341, 147.343, 25.853, -50.985, -16.964]
  MoveL 1467 to (-52.16, 198.42, -5) mm, rotated rx 180 ry 0 rz -179 deg; joints [13.966, -74.548, 120.871, 18.977, -47.919, -12.977]
  MoveC 1468 to (-51.71, 198.23, -5) mm, rotated rx 180 ry 0 rz -179 deg; joints [13.97, -74.52, 120.834, 18.984, -47.911, -12.985] to (-51.52, 197.78, -5) mm, rotated rx -180 ry 0 rz -179 deg; joints [13.988, -74.504, 120.812, 19.01, -47.91, -13.003]
  MoveL 1469 to (-51.52, 197.15, -5) mm, rotated rx -180 ry 0 rz -179 deg; joints [14.016, -74.495, 120.801, 19.048, -47.914, -13.029]
  MoveC 1470 to (-51.52, 196.7, -4.81) mm, rotated rx 180 ry 0 rz -179 deg; joints [14.037, -74.498, 120.788, 19.079, -47.904, -13.054] to (-51.52, 196.52, -4.37) mm, rotated rx 180 ry 0 rz -179 deg; joints [14.045, -74.514, 120.772, 19.099, -47.875, -13.075]
  Set speed (500.0 mm/s)
  MoveL 1471 to (-51.52, 196.52, 5) mm, rotated rx -180 ry 0 rz -179 deg; joints [14.045, -74.91, 120.503, 19.299, -47.248, -13.371]
  MoveL 1472 to (-52.79, 196.52, 5) mm, rotated rx -180 ry 0 rz -179 deg; joints [14.058, -74.982, 120.599, 19.309, -47.273, -13.373]
  Set speed (25.4 mm/s)
  MoveL 1473 to (-52.79, 196.52, 1) mm, rotated rx -180 ry 0 rz -179 deg; joints [14.058, -74.814, 120.715, 19.223, -47.541, -13.245]
  MoveL 1474 to (-52.79, 196.52, -7.72) mm, rotated rx 180 ry 0 rz -179 deg; joints [14.058, -74.443, 120.962, 19.039, -48.126, -12.972]
  MoveC 1475 to (-52.79, 196.7, -8.16) mm, rotated rx -180 ry 0 rz -179 deg; joints [14.05, -74.426, 120.978, 19.019, -48.155, -12.95] to (-52.79, 197.15, -8.35) mm, rotated rx -180 ry 0 rz -179 deg; joints [14.03, -74.424, 120.991, 18.988, -48.165, -12.926]
  Set speed (50.8 mm/s)
  MoveL 1476 to (-52.79, 197.79, -8.35) mm, rotated rx 180 ry 0 rz -179 deg; joints [14.001, -74.432, 121.002, 18.95, -48.161, -12.9]
  MoveC 1477 to (-52.61, 198.23, -8.35) mm, rotated rx -180 ry 0 rz -179 deg; joints [13.979, -74.427, 120.996, 18.922, -48.154, -12.882] to (-52.16, 198.42, -8.35) mm, rotated rx -180 ry 0 rz -179 deg; joints [13.966, -74.405, 120.965, 18.907, -48.144, -12.874]
  MoveL 1478 to (-14.06, 198.42, -8.35) mm, rotated rx -180 ry 0 rz -179 deg; joints [13.585, -72.259, 118.042, 18.632, -47.323, -12.874]
  MoveL 1479 to (-14.06, 350.82, -8.35) mm, rotated rx -180 ry 0 rz -179 deg; joints [6.808, -73.666, 119.969, 9.376, -46.688, -6.462]
  MoveL 1480 to (-39.46, 350.82, -8.35) mm, rotated rx -180 ry 0 rz -179 deg; joints [6.927, -75.131, 121.935, 9.461, -47.195, -6.461]
  MoveC 1481 to (-52.16, 338.12, -8.35) mm, rotated rx 180 ry 0 rz -179 deg; joints [7.58, -75.786, 122.8, 10.31, -47.478, -7.009] to (-64.86, 350.82, -8.35) mm, rotated rx 180 ry 0 rz -179 deg; joints [7.051, -76.607, 123.871, 9.559, -47.663, -6.471]
  MoveL 1482 to (-90.26, 350.82, -8.35) mm, rotated rx -180 ry 0 rz -179 deg; joints [7.181, -78.096, 125.779, 9.669, -48.091, -6.493]
  MoveL 1483 to (-166.46, 350.82, -8.35) mm, rotated rx -180 ry 0 rz -179 deg; joints [7.604, -82.666, 131.341, 10.081, -49.116, -6.637]
  MoveC 1484 to (-179.16, 338.12, -8.35) mm, rotated rx -180 ry 0 rz -179 deg; joints [8.339, -83.35, 132.134, 11.027, -49.312, -7.24] to (-191.86, 350.82, -8.35) mm, rotated rx -180 ry 0 rz -179 deg; joints [7.759, -84.233, 133.142, 10.248, -49.364, -6.715]
  MoveL 1485 to (-293.46, 350.82, -8.35) mm, rotated rx 180 ry 0 rz -179 deg; joints [8.456, -90.809, 140.091, 11.098, -49.816, -7.213]
  MoveC 1486 to (-306.16, 338.12, -8.35) mm, rotated rx 180 ry 0 rz -179 deg; joints [9.296, -91.552, 140.814, 12.19, -49.907, -7.92] to (-318.86, 350.82, -8.35) mm, rotated rx -180 ry 0 rz -179 deg; joints [8.653, -92.548, 141.763, 11.365, -49.775, -7.396]
  MoveL 1487 to (-395.06, 350.82, -8.35) mm, rotated rx -180 ry 0 rz -179 deg; joints [9.312, -98.072, 146.618, 12.341, -49.209, -8.135]
  MoveL 1488 to (-420.46, 350.82, -8.35) mm, rotated rx 180 ry 0 rz -179 deg; joints [9.558, -100.035, 148.178, 12.739, -48.852, -8.461]
  MoveC 1489 to (-433.16, 338.12, -8.35) mm, rotated rx -180 ry 0 rz -179 deg; joints [10.536, -100.879, 148.824, 14.063, -48.81, -9.367] to (-445.86, 350.82, -8.35) mm, rotated rx -180 ry 0 rz -179 deg; joints [9.818, -102.068, 149.707, 13.181, -48.4, -8.838]
  MoveL 1490 to (-471.26, 350.82, -8.35) mm, rotated rx 180 ry 0 rz -179 deg; joints [10.095, -104.18, 151.204, 13.676, -47.845, -9.275]
  MoveL 1491 to (-471.26, 198.42, -8.35) mm, rotated rx -180 ry 0 rz -179 deg; joints [20.36, -101.045, 148.949, 26.57, -51.061, -17.449]
  MoveL 1492 to (-445.86, 198.42, -8.35) mm, rotated rx -180 ry 0 rz -179 deg; joints [19.804, -99.135, 147.473, 25.735, -51.287, -16.776]
  MoveL 1493 to (-52.16, 198.42, -8.35) mm, rotated rx -180 ry 0 rz -179 deg; joints [13.966, -74.405, 120.965, 18.907, -48.144, -12.874]
  MoveC 1494 to (-51.71, 198.23, -8.35) mm, rotated rx -180 ry 0 rz -179 deg; joints [13.97, -74.377, 120.928, 18.915, -48.136, -12.881] to (-51.52, 197.79, -8.35) mm, rotated rx -180 ry 0 rz -179 deg; joints [13.988, -74.36, 120.906, 18.94, -48.135, -12.899]
  MoveL 1495 to (-51.52, 197.15, -8.35) mm, rotated rx 180 ry 0 rz -179 deg; joints [14.016, -74.352, 120.895, 18.978, -48.138, -12.925]
  MoveC 1496 to (-51.52, 196.7, -8.16) mm, rotated rx -180 ry 0 rz -179 deg; joints [14.037, -74.354, 120.882, 19.009, -48.129, -12.95] to (-51.52, 196.52, -7.72) mm, rotated rx -180 ry 0 rz -179 deg; joints [14.045, -74.371, 120.866, 19.029, -48.1, -12.971]
  Set speed (500.0 mm/s)
  MoveL 1497 to (-51.52, 196.51, 6) mm, rotated rx -180 ry 0 rz -179 deg; joints [14.045, -74.951, 120.474, 19.321, -47.181, -13.403]
  MoveL 1498 to (18.41, 196.52, 6) mm, rotated rx -180 ry 0 rz -179 deg; joints [13.358, -70.985, 115.064, 18.847, -45.657, -13.419]
  Set speed (25.4 mm/s)
  MoveL 1499 to (18.41, 196.52, -4.36) mm, rotated rx 180 ry 0 rz -179 deg; joints [13.358, -70.576, 115.352, 18.631, -46.318, -13.107]
  MoveC 1500 to (18.41, 196.7, -4.81) mm, rotated rx -180 ry 0 rz -179 deg; joints [13.35, -70.56, 115.368, 18.611, -46.346, -13.086] to (18.41, 197.15, -5) mm, rotated rx -180 ry 0 rz -179 deg; joints [13.331, -70.558, 115.381, 18.581, -46.356, -13.062]
  Set speed (50.8 mm/s)
  MoveL 1501 to (18.41, 197.78, -5) mm, rotated rx -180 ry 0 rz -179 deg; joints [13.304, -70.566, 115.392, 18.543, -46.353, -13.036]
  MoveC 1502 to (18.6, 198.23, -5) mm, rotated rx -180 ry 0 rz -179 deg; joints [13.283, -70.561, 115.385, 18.516, -46.346, -13.017] to (19.05, 198.42, -5) mm, rotated rx 180 ry 0 rz -179 deg; joints [13.271, -70.538, 115.352, 18.502, -46.334, -13.01]
  MoveL 1503 to (39.46, 198.42, -5) mm, rotated rx -180 ry 0 rz -179 deg; joints [13.085, -69.394, 113.722, 18.399, -45.832, -13.049]
  MoveL 1504 to (471.26, 198.42, -5) mm, rotated rx -180 ry 0 rz -179 deg; joints [10.144, -43.242, 71.171, 20.906, -29.574, -18.377]
  MoveL 1505 to (471.26, 350.82, -5) mm, rotated rx -180 ry 0 rz -179 deg; joints [5.194, -44.522, 73.443, 10.645, -29.345, -9.305]
  MoveL 1506 to (445.86, 350.82, -5) mm, rotated rx -180 ry 0 rz -179 deg; joints [5.256, -46.297, 76.569, 10.342, -30.682, -8.919]
  MoveC 1507 to (433.16, 338.12, -5) mm, rotated rx -180 ry 0 rz -179 deg; joints [5.713, -47.096, 77.965, 11.033, -31.342, -9.454] to (420.46, 350.82, -5) mm, rotated rx -180 ry 0 rz -179 deg; joints [5.32, -48.017, 79.567, 10.09, -31.95, -8.587]
  MoveL 1508 to (395.06, 350.82, -5) mm, rotated rx -180 ry 0 rz -179 deg; joints [5.385, -49.69, 82.453, 9.882, -33.154, -8.298]
  MoveL 1509 to (318.86, 350.82, -5) mm, rotated rx -180 ry 0 rz -179 deg; joints [5.595, -54.488, 90.555, 9.448, -36.44, -7.625]
  MoveC 1510 to (306.16, 338.12, -5) mm, rotated rx -180 ry 0 rz -179 deg; joints [6.091, -55.197, 91.728, 10.163, -36.965, -8.151] to (293.46, 350.82, -5) mm, rotated rx -180 ry 0 rz -179 deg; joints [5.67, -56.031, 93.1, 9.352, -37.439, -7.45]
  MoveL 1511 to (191.86, 350.82, -5) mm, rotated rx -180 ry 0 rz -179 deg; joints [5.993, -62.016, 102.673, 9.153, -41.021, -6.931]
  MoveC 1512 to (179.16, 338.12, -5) mm, rotated rx 180 ry 0 rz -179 deg; joints [6.535, -62.681, 103.706, 9.9, -41.451, -7.453] to (166.46, 350.82, -5) mm, rotated rx 180 ry 0 rz -179 deg; joints [6.081, -63.48, 104.937, 9.141, -41.82, -6.838]
  MoveL 1513 to (90.26, 350.82, -5) mm, rotated rx -180 ry 0 rz -179 deg; joints [6.364, -67.839, 111.47, 9.182, -44, -6.632]
  MoveL 1514 to (64.86, 350.82, -5) mm, rotated rx 180 ry 0 rz -179 deg; joints [6.466, -69.288, 113.57, 9.22, -44.655, -6.587]
  MoveC 1515 to (61.14, 341.84, -5) mm, rotated rx 180 ry 0 rz -179 deg; joints [6.864, -69.449, 113.801, 9.771, -44.771, -6.97] to (52.16, 338.12, -5) mm, rotated rx 180 ry 0 rz -179 deg; joints [7.064, -69.939, 114.502, 10.015, -45.003, -7.117]
  MoveL 1516 to (52.16, 338.12, -5) mm, rotated rx -180 ry 0 rz -179 deg; joints [7.064, -69.939, 114.502, 10.015, -45.003, -7.117]
  MoveC 1517 to (43.18, 341.84, -5) mm, rotated rx 180 ry 0 rz -179 deg; joints [6.944, -70.473, 115.261, 9.809, -45.209, -6.945] to (39.46, 350.82, -5) mm, rotated rx 180 ry 0 rz -179 deg; joints [6.571, -70.738, 115.634, 9.27, -45.273, -6.552]
  MoveL 1518 to (14.06, 350.82, -5) mm, rotated rx -180 ry 0 rz -179 deg; joints [6.681, -72.192, 117.665, 9.331, -45.855, -6.528]
  MoveL 1519 to (14.06, 198.42, -5) mm, rotated rx -180 ry 0 rz -179 deg; joints [13.318, -70.818, 115.747, 18.53, -46.454, -13.003]
  MoveL 1520 to (19.05, 198.42, -5) mm, rotated rx -180 ry 0 rz -179 deg; joints [13.271, -70.538, 115.352, 18.502, -46.334, -13.01]
  MoveC 1521 to (19.49, 198.23, -5) mm, rotated rx -180 ry 0 rz -179 deg; joints [13.275, -70.511, 115.314, 18.511, -46.324, -13.019] to (19.68, 197.79, -5) mm, rotated rx -180 ry 0 rz -179 deg; joints [13.292, -70.495, 115.291, 18.536, -46.322, -13.038]
  MoveL 1522 to (19.68, 197.15, -5) mm, rotated rx -180 ry 0 rz -179 deg; joints [13.319, -70.487, 115.28, 18.574, -46.325, -13.064]
  MoveC 1523 to (19.68, 196.7, -4.81) mm, rotated rx -180 ry 0 rz -179 deg; joints [13.338, -70.489, 115.267, 18.604, -46.315, -13.088] to (19.68, 196.52, -4.37) mm, rotated rx -180 ry 0 rz -179 deg; joints [13.346, -70.504, 115.252, 18.624, -46.288, -13.109]
  Set speed (500.0 mm/s)
  MoveL 1524 to (19.68, 196.52, 5) mm, rotated rx 180 ry 0 rz -179 deg; joints [13.346, -70.874, 114.991, 18.819, -45.691, -13.391]
  MoveL 1525 to (18.41, 196.52, 5) mm, rotated rx 180 ry 0 rz -179 deg; joints [13.358, -70.946, 115.092, 18.826, -45.721, -13.389]
  Set speed (25.4 mm/s)
  MoveL 1526 to (18.41, 196.52, 1) mm, rotated rx -180 ry 0 rz -179 deg; joints [13.358, -70.788, 115.204, 18.742, -45.976, -13.268]
  MoveL 1527 to (18.41, 196.52, -7.71) mm, rotated rx 180 ry 0 rz -179 deg; joints [13.358, -70.442, 115.444, 18.562, -46.532, -13.008]
  MoveC 1528 to (18.41, 196.7, -8.16) mm, rotated rx -180 ry 0 rz -179 deg; joints [13.35, -70.426, 115.459, 18.542, -46.56, -12.987] to (18.41, 197.15, -8.35) mm, rotated rx 180 ry 0 rz -179 deg; joints [13.331, -70.424, 115.472, 18.512, -46.569, -12.963]
  Set speed (50.8 mm/s)
  MoveL 1529 to (18.41, 197.79, -8.35) mm, rotated rx 180 ry 0 rz -179 deg; joints [13.304, -70.432, 115.483, 18.475, -46.566, -12.937]
  MoveC 1530 to (18.6, 198.23, -8.35) mm, rotated rx -180 ry 0 rz -179 deg; joints [13.283, -70.427, 115.476, 18.448, -46.56, -12.919] to (19.04, 198.42, -8.35) mm, rotated rx 180 ry 0 rz -179 deg; joints [13.271, -70.404, 115.444, 18.435, -46.548, -12.912]
  MoveL 1531 to (39.46, 198.42, -8.35) mm, rotated rx 180 ry 0 rz -179 deg; joints [13.085, -69.262, 113.813, 18.331, -46.042, -12.952]
  MoveL 1532 to (471.26, 198.42, -8.35) mm, rotated rx -180 ry 0 rz -179 deg; joints [10.144, -43.162, 71.271, 20.793, -29.743, -18.248]
  MoveL 1533 to (471.26, 350.82, -8.35) mm, rotated rx -180 ry 0 rz -179 deg; joints [5.194, -44.439, 73.542, 10.586, -29.522, -9.237]
  MoveL 1534 to (445.86, 350.82, -8.35) mm, rotated rx 180 ry 0 rz -179 deg; joints [5.256, -46.212, 76.665, 10.287, -30.861, -8.856]
  MoveC 1535 to (433.16, 338.12, -8.35) mm, rotated rx 180 ry 0 rz -179 deg; joints [5.713, -47.009, 78.06, 10.976, -31.521, -9.388] to (420.46, 350.82, -8.35) mm, rotated rx 180 ry 0 rz -179 deg; joints [5.32, -47.928, 79.661, 10.039, -32.13, -8.526]
  MoveL 1536 to (395.06, 350.82, -8.35) mm, rotated rx -180 ry 0 rz -179 deg; joints [5.385, -49.598, 82.545, 9.834, -33.335, -8.24]
  MoveL 1537 to (318.86, 350.82, -8.35) mm, rotated rx -180 ry 0 rz -179 deg; joints [5.595, -54.387, 90.644, 9.406, -36.627, -7.572]
  MoveC 1538 to (306.16, 338.12, -8.35) mm, rotated rx -180 ry 0 rz -179 deg; joints [6.091, -55.095, 91.817, 10.119, -37.154, -8.095] to (293.46, 350.82, -8.35) mm, rotated rx -180 ry 0 rz -179 deg; joints [5.67, -55.927, 93.189, 9.312, -37.629, -7.399]
  MoveL 1539 to (191.86, 350.82, -8.35) mm, rotated rx -180 ry 0 rz -179 deg; joints [5.993, -61.9, 102.762, 9.116, -41.222, -6.882]
  MoveC 1540 to (179.16, 338.12, -8.35) mm, rotated rx -180 ry 0 rz -179 deg; joints [6.535, -62.564, 103.795, 9.86, -41.653, -7.4] to (166.46, 350.82, -8.35) mm, rotated rx -180 ry 0 rz -179 deg; joints [6.081, -63.362, 105.025, 9.105, -42.025, -6.789]
  MoveL 1541 to (90.26, 350.82, -8.35) mm, rotated rx 180 ry 0 rz -179 deg; joints [6.364, -67.711, 111.56, 9.146, -44.215, -6.583]
  MoveL 1542 to (64.86, 350.82, -8.35) mm, rotated rx -180 ry 0 rz -179 deg; joints [6.466, -69.156, 113.66, 9.184, -44.874, -6.536]
  MoveC 1543 to (61.14, 341.84, -8.35) mm, rotated rx -180 ry 0 rz -179 deg; joints [6.864, -69.317, 113.892, 9.733, -44.99, -6.917] to (52.16, 338.12, -8.35) mm, rotated rx -180 ry 0 rz -179 deg; joints [7.064, -69.806, 114.593, 9.976, -45.223, -7.063]
  MoveL 1544 to (52.16, 338.12, -8.35) mm, rotated rx 180 ry 0 rz -179 deg; joints [7.064, -69.806, 114.593, 9.976, -45.223, -7.063]
  MoveC 1545 to (43.18, 341.84, -8.35) mm, rotated rx -180 ry 0 rz -179 deg; joints [6.944, -70.34, 115.352, 9.771, -45.431, -6.891] to (39.46, 350.82, -8.35) mm, rotated rx 180 ry 0 rz -179 deg; joints [6.571, -70.603, 115.726, 9.234, -45.496, -6.501]
  MoveL 1546 to (14.06, 350.82, -8.35) mm, rotated rx -180 ry 0 rz -179 deg; joints [6.681, -72.054, 117.757, 9.295, -46.082, -6.477]
  MoveL 1547 to (14.06, 198.42, -8.35) mm, rotated rx -180 ry 0 rz -179 deg; joints [13.318, -70.683, 115.839, 18.462, -46.668, -12.904]
  MoveL 1548 to (19.04, 198.42, -8.35) mm, rotated rx 180 ry 0 rz -179 deg; joints [13.271, -70.404, 115.444, 18.435, -46.548, -12.912]
  MoveC 1549 to (19.49, 198.23, -8.35) mm, rotated rx -180 ry 0 rz -179 deg; joints [13.275, -70.377, 115.405, 18.443, -46.538, -12.92] to (19.68, 197.79, -8.35) mm, rotated rx -180 ry 0 rz -179 deg; joints [13.292, -70.361, 115.382, 18.468, -46.535, -12.939]
  MoveL 1550 to (19.68, 197.15, -8.35) mm, rotated rx -180 ry 0 rz -179 deg; joints [13.319, -70.353, 115.371, 18.506, -46.538, -12.965]
  MoveC 1551 to (19.68, 196.7, -8.16) mm, rotated rx -180 ry 0 rz -179 deg; joints [13.338, -70.355, 115.359, 18.536, -46.529, -12.989] to (19.68, 196.52, -7.72) mm, rotated rx -180 ry 0 rz -179 deg; joints [13.346, -70.371, 115.343, 18.556, -46.501, -13.01]
  Set speed (500.0 mm/s)
  MoveL 1552 to (19.68, 196.52, 6) mm, rotated rx 180 ry 0 rz -179 deg; joints [13.346, -70.913, 114.963, 18.84, -45.627, -13.421]
  MoveL 1553 to (18.41, 382.85, 6) mm, rotated rx -180 ry 0 rz -179 deg; joints [5.246, -72.547, 117.231, 7.439, -44.926, -5.282]
  Set speed (25.4 mm/s)
  MoveL 1554 to (18.41, 382.85, -4.37) mm, rotated rx -180 ry 0 rz -179 deg; joints [5.246, -72.127, 117.523, 7.348, -45.632, -5.153]
  MoveC 1555 to (18.41, 383.04, -4.81) mm, rotated rx 180 ry 0 rz -179 deg; joints [5.238, -72.11, 117.536, 7.333, -45.662, -5.139] to (18.41, 383.49, -5) mm, rotated rx -180 ry 0 rz -179 deg; joints [5.218, -72.104, 117.544, 7.304, -45.673, -5.118]
  Set speed (50.8 mm/s)
  MoveL 1556 to (18.41, 384.12, -5) mm, rotated rx -180 ry 0 rz -179 deg; joints [5.19, -72.107, 117.548, 7.264, -45.672, -5.09]
  MoveC 1557 to (18.6, 384.57, -5) mm, rotated rx -180 ry 0 rz -179 deg; joints [5.169, -72.098, 117.535, 7.236, -45.667, -5.071] to (19.04, 384.76, -5) mm, rotated rx -180 ry 0 rz -179 deg; joints [5.16, -72.073, 117.501, 7.224, -45.656, -5.063]
  MoveL 1558 to (64.86, 384.76, -5) mm, rotated rx -180 ry 0 rz -179 deg; joints [5.017, -69.448, 113.801, 7.158, -44.576, -5.112]
  MoveL 1559 to (471.26, 384.76, -5) mm, rotated rx 180 ry 0 rz -179 deg; joints [4.08, -44.675, 73.715, 8.36, -29.3, -7.303]
  MoveL 1560 to (471.26, 537.16, -5) mm, rotated rx 180 ry 0 rz -179 deg; joints [-0.936, -44.783, 73.906, -1.924, -29.136, 1.68]
  MoveL 1561 to (445.86, 537.16, -5) mm, rotated rx -180 ry 0 rz -179 deg; joints [-0.965, -46.554, 77.018, -1.903, -30.479, 1.64]
  MoveC 1562 to (433.16, 524.46, -5) mm, rotated rx -180 ry 0 rz -179 deg; joints [-0.552, -47.445, 78.573, -1.068, -31.132, 0.915] to (420.46, 537.16, -5) mm, rotated rx 180 ry 0 rz -179 deg; joints [-0.995, -48.27, 80.005, -1.89, -31.749, 1.608]
  MoveL 1563 to (395.06, 537.16, -5) mm, rotated rx -180 ry 0 rz -179 deg; joints [-1.025, -49.94, 82.882, -1.885, -32.956, 1.581]
  MoveL 1564 to (318.86, 537.16, -5) mm, rotated rx -180 ry 0 rz -179 deg; joints [-1.122, -54.735, 90.964, -1.898, -36.244, 1.531]
  MoveC 1565 to (306.16, 524.46, -5) mm, rotated rx 180 ry 0 rz -179 deg; joints [-0.678, -55.535, 92.286, -1.132, -36.756, 0.907] to (293.46, 537.16, -5) mm, rotated rx 180 ry 0 rz -179 deg; joints [-1.157, -56.278, 93.505, -1.912, -37.243, 1.522]
  MoveL 1566 to (191.86, 537.16, -5) mm, rotated rx -180 ry 0 rz -179 deg; joints [-1.307, -62.27, 103.068, -1.999, -40.816, 1.513]
  MoveC 1567 to (179.16, 524.46, -5) mm, rotated rx -180 ry 0 rz -179 deg; joints [-0.825, -63.031, 104.246, -1.252, -41.222, 0.941] to (166.46, 537.16, -5) mm, rotated rx -180 ry 0 rz -179 deg; joints [-1.347, -63.737, 105.331, -2.029, -41.611, 1.518]
  MoveL 1568 to (90.26, 537.16, -5) mm, rotated rx 180 ry 0 rz -179 deg; joints [-1.479, -68.108, 111.863, -2.138, -43.775, 1.544]
  MoveL 1569 to (64.86, 537.16, -5) mm, rotated rx -180 ry 0 rz -179 deg; joints [-1.526, -69.562, 113.964, -2.181, -44.422, 1.558]
  MoveC 1570 to (61.14, 528.18, -5) mm, rotated rx -180 ry 0 rz -179 deg; joints [-1.147, -69.796, 114.298, -1.636, -44.514, 1.167] to (52.16, 524.46, -5) mm, rotated rx 180 ry 0 rz -179 deg; joints [-1, -70.319, 115.042, -1.421, -44.732, 1.01]
  MoveL 1571 to (52.16, 524.46, -5) mm, rotated rx 180 ry 0 rz -179 deg; joints [-1, -70.319, 115.042, -1.421, -44.732, 1.01]
  MoveC 1572 to (43.18, 528.18, -5) mm, rotated rx -180 ry 0 rz -179 deg; joints [-1.176, -70.826, 115.759, -1.665, -44.945, 1.179] to (39.46, 537.16, -5) mm, rotated rx -180 ry 0 rz -179 deg; joints [-1.575, -71.018, 116.029, -2.227, -45.033, 1.574]
  MoveL 1573 to (14.06, 537.16, -5) mm, rotated rx -180 ry 0 rz -179 deg; joints [-1.626, -72.479, 118.061, -2.276, -45.605, 1.593]
  MoveL 1574 to (14.06, 384.76, -5) mm, rotated rx -180 ry 0 rz -179 deg; joints [5.176, -72.36, 117.897, 7.233, -45.767, -5.059]
  MoveL 1575 to (19.04, 384.76, -5) mm, rotated rx -180 ry 0 rz -179 deg; joints [5.16, -72.073, 117.501, 7.224, -45.656, -5.063]
  MoveC 1576 to (19.49, 384.57, -5) mm, rotated rx -180 ry 0 rz -179 deg; joints [5.166, -72.046, 117.464, 7.235, -45.647, -5.071] to (19.68, 384.12, -5) mm, rotated rx -180 ry 0 rz -179 deg; joints [5.186, -72.034, 117.447, 7.262, -45.644, -5.091]
  MoveL 1577 to (19.68, 383.49, -5) mm, rotated rx 180 ry 0 rz -179 deg; joints [5.214, -72.031, 117.443, 7.301, -45.645, -5.119]
  MoveC 1578 to (19.68, 383.04, -4.81) mm, rotated rx 180 ry 0 rz -179 deg; joints [5.234, -72.037, 117.435, 7.331, -45.633, -5.14] to (19.68, 382.85, -4.37) mm, rotated rx -180 ry 0 rz -179 deg; joints [5.242, -72.054, 117.422, 7.346, -45.603, -5.154]
  Set speed (500.0 mm/s)
  MoveL 1579 to (19.68, 382.85, 5) mm, rotated rx -180 ry 0 rz -179 deg; joints [5.242, -72.434, 117.158, 7.428, -44.966, -5.27]
  MoveL 1580 to (18.41, 382.85, 5) mm, rotated rx -180 ry 0 rz -179 deg; joints [5.246, -72.507, 117.259, 7.43, -44.994, -5.269]
  Set speed (25.4 mm/s)
  MoveL 1581 to (18.41, 382.85, 1) mm, rotated rx -180 ry 0 rz -179 deg; joints [5.246, -72.346, 117.373, 7.395, -45.266, -5.219]
  MoveL 1582 to (18.41, 382.85, -7.72) mm, rotated rx -180 ry 0 rz -179 deg; joints [5.246, -71.99, 117.615, 7.32, -45.86, -5.112]
  MoveC 1583 to (18.41, 383.04, -8.16) mm, rotated rx -180 ry 0 rz -179 deg; joints [5.238, -71.972, 117.629, 7.304, -45.89, -5.098] to (18.41, 383.49, -8.35) mm, rotated rx -180 ry 0 rz -179 deg; joints [5.218, -71.966, 117.636, 7.275, -45.901, -5.077]
  Set speed (50.8 mm/s)
  MoveL 1584 to (18.41, 384.12, -8.35) mm, rotated rx 180 ry 0 rz -179 deg; joints [5.19, -71.969, 117.64, 7.236, -45.9, -5.049]
  MoveC 1585 to (18.6, 384.57, -8.35) mm, rotated rx 180 ry 0 rz -179 deg; joints [5.169, -71.96, 117.628, 7.208, -45.895, -5.03] to (19.04, 384.76, -8.35) mm, rotated rx -180 ry 0 rz -179 deg; joints [5.16, -71.935, 117.593, 7.196, -45.884, -5.023]
  MoveL 1586 to (64.86, 384.76, -8.35) mm, rotated rx -180 ry 0 rz -179 deg; joints [5.017, -69.317, 113.891, 7.13, -44.797, -5.072]
  MoveL 1587 to (471.26, 384.76, -8.35) mm, rotated rx -180 ry 0 rz -179 deg; joints [4.08, -44.592, 73.813, 8.314, -29.479, -7.25]
  MoveL 1588 to (471.26, 537.16, -8.35) mm, rotated rx -180 ry 0 rz -179 deg; joints [-0.936, -44.7, 74.004, -1.913, -29.317, 1.668]
  MoveL 1589 to (445.86, 537.16, -8.35) mm, rotated rx -180 ry 0 rz -179 deg; joints [-0.965, -46.468, 77.114, -1.893, -30.66, 1.628]
  MoveC 1590 to (433.16, 524.46, -8.35) mm, rotated rx 180 ry 0 rz -179 deg; joints [-0.552, -47.357, 78.667, -1.063, -31.315, 0.908] to (420.46, 537.16, -8.35) mm, rotated rx 180 ry 0 rz -179 deg; joints [-0.995, -48.181, 80.099, -1.881, -31.932, 1.596]
  MoveL 1591 to (395.06, 537.16, -8.35) mm, rotated rx 180 ry 0 rz -179 deg; joints [-1.025, -49.848, 82.974, -1.875, -33.14, 1.57]
  MoveL 1592 to (318.86, 537.16, -8.35) mm, rotated rx -180 ry 0 rz -179 deg; joints [-1.122, -54.634, 91.053, -1.89, -36.434, 1.521]
  MoveC 1593 to (306.16, 524.46, -8.35) mm, rotated rx -180 ry 0 rz -179 deg; joints [-0.678, -55.432, 92.374, -1.127, -36.948, 0.901] to (293.46, 537.16, -8.35) mm, rotated rx -180 ry 0 rz -179 deg; joints [-1.157, -56.174, 93.594, -1.903, -37.435, 1.511]
  MoveL 1594 to (191.86, 537.16, -8.35) mm, rotated rx 180 ry 0 rz -179 deg; joints [-1.307, -62.154, 103.156, -1.991, -41.02, 1.503]
  MoveC 1595 to (179.16, 524.46, -8.35) mm, rotated rx 180 ry 0 rz -179 deg; joints [-0.825, -62.913, 104.335, -1.246, -41.428, 0.935] to (166.46, 537.16, -8.35) mm, rotated rx -180 ry 0 rz -179 deg; joints [-1.347, -63.618, 105.419, -2.021, -41.819, 1.507]
  MoveL 1596 to (90.26, 537.16, -8.35) mm, rotated rx -180 ry 0 rz -179 deg; joints [-1.479, -67.98, 111.953, -2.13, -43.993, 1.532]
  MoveL 1597 to (64.86, 537.16, -8.35) mm, rotated rx -180 ry 0 rz -179 deg; joints [-1.526, -69.43, 114.054, -2.172, -44.645, 1.546]
  MoveC 1598 to (61.14, 528.18, -8.35) mm, rotated rx -180 ry 0 rz -179 deg; joints [-1.147, -69.664, 114.389, -1.629, -44.737, 1.158] to (52.16, 524.46, -8.35) mm, rotated rx 180 ry 0 rz -179 deg; joints [-1, -70.185, 115.133, -1.416, -44.956, 1.002]
  MoveL 1599 to (52.16, 524.46, -8.35) mm, rotated rx -180 ry 0 rz -179 deg; joints [-1, -70.185, 115.133, -1.416, -44.956, 1.002]
  MoveC 1600 to (43.18, 528.18, -8.35) mm, rotated rx -180 ry 0 rz -179 deg; joints [-1.176, -70.691, 115.85, -1.658, -45.171, 1.169] to (39.46, 537.16, -8.35) mm, rotated rx -180 ry 0 rz -179 deg; joints [-1.575, -70.883, 116.121, -2.218, -45.259, 1.562]
  MoveL 1601 to (14.06, 537.16, -8.35) mm, rotated rx -180 ry 0 rz -179 deg; joints [-1.626, -72.34, 118.154, -2.267, -45.836, 1.58]
  MoveL 1602 to (14.06, 384.76, -8.35) mm, rotated rx -180 ry 0 rz -179 deg; joints [5.176, -72.221, 117.99, 7.205, -45.995, -5.019]
  MoveL 1603 to (19.04, 384.76, -8.35) mm, rotated rx 180 ry 0 rz -179 deg; joints [5.16, -71.935, 117.593, 7.196, -45.884, -5.023]
  MoveC 1604 to (19.49, 384.57, -8.35) mm, rotated rx -180 ry 0 rz -179 deg; joints [5.166, -71.909, 117.556, 7.206, -45.875, -5.031] to (19.68, 384.12, -8.35) mm, rotated rx -180 ry 0 rz -179 deg; joints [5.186, -71.896, 117.539, 7.234, -45.871, -5.05]
  MoveL 1605 to (19.68, 383.49, -8.35) mm, rotated rx 180 ry 0 rz -179 deg; joints [5.214, -71.894, 117.535, 7.273, -45.873, -5.078]
  MoveC 1606 to (19.68, 383.04, -8.16) mm, rotated rx -180 ry 0 rz -179 deg; joints [5.234, -71.899, 117.527, 7.302, -45.861, -5.099] to (19.68, 382.85, -7.72) mm, rotated rx -180 ry 0 rz -179 deg; joints [5.242, -71.917, 117.514, 7.317, -45.831, -5.113]
  Set speed (500.0 mm/s)
  MoveL 1607 to (19.68, 382.85, 6) mm, rotated rx 180 ry 0 rz -179 deg; joints [5.242, -72.474, 117.13, 7.437, -44.898, -5.283]
  MoveL 1608 to (-12.15, 384.12, 6) mm, rotated rx -180 ry 0 rz -179 deg; joints [5.291, -74.327, 119.642, 7.422, -45.556, -5.211]
  Set speed (25.4 mm/s)
  MoveL 1609 to (-12.15, 384.12, -4.36) mm, rotated rx -180 ry 0 rz -179 deg; joints [5.291, -73.894, 119.938, 7.331, -46.279, -5.081]
  MoveC 1610 to (-12.34, 384.12, -4.81) mm, rotated rx -180 ry 0 rz -179 deg; joints [5.292, -73.886, 119.966, 7.328, -46.314, -5.076] to (-12.79, 384.12, -5) mm, rotated rx -180 ry 0 rz -179 deg; joints [5.293, -73.904, 120.006, 7.327, -46.336, -5.073]
  Set speed (50.8 mm/s)
  MoveL 1611 to (-13.42, 384.12, -5) mm, rotated rx -180 ry 0 rz -179 deg; joints [5.296, -73.941, 120.055, 7.328, -46.349, -5.073]
  MoveC 1612 to (-13.87, 384.31, -5) mm, rotated rx 180 ry 0 rz -179 deg; joints [5.289, -73.968, 120.092, 7.318, -46.358, -5.065] to (-14.06, 384.76, -5) mm, rotated rx 180 ry 0 rz -179 deg; joints [5.269, -73.98, 120.109, 7.29, -46.361, -5.045]
  MoveL 1613 to (-14.06, 537.16, -5) mm, rotated rx -180 ry 0 rz -179 deg; joints [-1.685, -74.103, 120.274, -2.335, -46.195, 1.617]
  MoveL 1614 to (-39.46, 537.16, -5) mm, rotated rx 180 ry 0 rz -179 deg; joints [-1.74, -75.58, 122.24, -2.392, -46.685, 1.642]
  MoveC 1615 to (-52.16, 524.46, -5) mm, rotated rx -180 ry 0 rz -179 deg; joints [-1.172, -76.355, 123.254, -1.604, -46.911, 1.096] to (-64.86, 537.16, -5) mm, rotated rx -180 ry 0 rz -179 deg; joints [-1.798, -77.068, 124.178, -2.454, -47.136, 1.67]
  MoveL 1616 to (-90.26, 537.16, -5) mm, rotated rx -180 ry 0 rz -179 deg; joints [-1.858, -78.571, 126.087, -2.519, -47.544, 1.701]
  MoveL 1617 to (-166.46, 537.16, -5) mm, rotated rx 180 ry 0 rz -179 deg; joints [-2.056, -83.189, 131.653, -2.745, -48.496, 1.82]
  MoveC 1618 to (-179.16, 524.46, -5) mm, rotated rx 180 ry 0 rz -179 deg; joints [-1.425, -84.017, 132.601, -1.899, -48.6, 1.256] to (-191.86, 537.16, -5) mm, rotated rx 180 ry 0 rz -179 deg; joints [-2.128, -84.775, 133.456, -2.832, -48.715, 1.869]
  MoveL 1619 to (-293.46, 537.16, -5) mm, rotated rx -180 ry 0 rz -179 deg; joints [-2.453, -91.443, 140.412, -3.25, -49.014, 2.133]
  MoveC 1620 to (-306.16, 524.46, -5) mm, rotated rx 180 ry 0 rz -179 deg; joints [-1.744, -92.369, 141.298, -2.313, -48.951, 1.519] to (-318.86, 537.16, -5) mm, rotated rx -180 ry 0 rz -179 deg; joints [-2.545, -93.211, 142.086, -3.377, -48.924, 2.22]
  MoveL 1621 to (-395.06, 537.16, -5) mm, rotated rx 180 ry 0 rz -179 deg; joints [-2.854, -98.839, 146.944, -3.831, -48.168, 2.557]
  MoveL 1622 to (-420.46, 537.16, -5) mm, rotated rx 180 ry 0 rz -179 deg; joints [-2.969, -100.843, 148.505, -4.014, -47.732, 2.702]
  MoveC 1623 to (-433.16, 524.46, -5) mm, rotated rx -180 ry 0 rz -179 deg; joints [-2.161, -101.939, 149.322, -2.935, -47.421, 1.987] to (-445.86, 537.16, -5) mm, rotated rx 180 ry 0 rz -179 deg; joints [-3.091, -102.923, 150.035, -4.215, -47.189, 2.867]
  MoveL 1624 to (-471.26, 537.16, -5) mm, rotated rx -180 ry 0 rz -179 deg; joints [-3.221, -105.086, 151.531, -4.44, -46.531, 3.058]
  MoveL 1625 to (-471.26, 384.76, -5) mm, rotated rx -180 ry 0 rz -179 deg; joints [7.7, -104.798, 151.337, 10.552, -47.027, -7.237]
  MoveL 1626 to (-14.06, 384.76, -5) mm, rotated rx 180 ry 0 rz -179 deg; joints [5.269, -73.98, 120.109, 7.29, -46.361, -5.045]
  MoveC 1627 to (-13.61, 384.57, -5) mm, rotated rx 180 ry 0 rz -179 deg; joints [5.276, -73.954, 120.073, 7.301, -46.352, -5.053] to (-13.42, 384.12, -5) mm, rotated rx -180 ry 0 rz -179 deg; joints [5.296, -73.941, 120.055, 7.328, -46.349, -5.073]
  MoveL 1628 to (-13.42, 383.49, -5) mm, rotated rx -180 ry 0 rz -179 deg; joints [5.324, -73.938, 120.052, 7.368, -46.351, -5.101]
  MoveC 1629 to (-13.42, 383.04, -4.81) mm, rotated rx -180 ry 0 rz -179 deg; joints [5.345, -73.944, 120.044, 7.398, -46.339, -5.122] to (-13.42, 382.85, -4.37) mm, rotated rx -180 ry 0 rz -179 deg; joints [5.353, -73.962, 120.03, 7.413, -46.308, -5.136]
  Set speed (500.0 mm/s)
  MoveL 1630 to (-13.42, 382.85, 5) mm, rotated rx 180 ry 0 rz -179 deg; joints [5.353, -74.354, 119.763, 7.496, -45.655, -5.255]
  MoveL 1631 to (-12.15, 384.12, 5) mm, rotated rx -180 ry 0 rz -179 deg; joints [5.291, -74.286, 119.671, 7.413, -45.626, -5.199]
  Set speed (25.4 mm/s)
  MoveL 1632 to (-12.15, 384.12, 1) mm, rotated rx 180 ry 0 rz -179 deg; joints [5.291, -74.119, 119.786, 7.377, -45.905, -5.148]
  MoveL 1633 to (-12.15, 384.12, -7.72) mm, rotated rx 180 ry 0 rz -179 deg; joints [5.291, -73.753, 120.032, 7.302, -46.513, -5.04]
  MoveC 1634 to (-12.34, 384.12, -8.16) mm, rotated rx 180 ry 0 rz -179 deg; joints [5.292, -73.744, 120.059, 7.299, -46.548, -5.034] to (-12.79, 384.12, -8.35) mm, rotated rx -180 ry 0 rz -179 deg; joints [5.293, -73.762, 120.1, 7.298, -46.57, -5.032]
  Set speed (50.8 mm/s)
  MoveL 1635 to (-13.42, 384.12, -8.35) mm, rotated rx -180 ry 0 rz -179 deg; joints [5.296, -73.799, 120.149, 7.3, -46.583, -5.032]
  MoveC 1636 to (-13.87, 384.31, -8.35) mm, rotated rx 180 ry 0 rz -179 deg; joints [5.289, -73.826, 120.185, 7.289, -46.592, -5.023] to (-14.06, 384.76, -8.35) mm, rotated rx 180 ry 0 rz -179 deg; joints [5.269, -73.838, 120.202, 7.262, -46.595, -5.004]
  MoveL 1637 to (-14.06, 537.16, -8.35) mm, rotated rx -180 ry 0 rz -179 deg; joints [-1.685, -73.96, 120.367, -2.326, -46.431, 1.603]
  MoveL 1638 to (-39.46, 537.16, -8.35) mm, rotated rx -180 ry 0 rz -179 deg; joints [-1.74, -75.434, 122.335, -2.383, -46.926, 1.628]
  MoveC 1639 to (-52.16, 524.46, -8.35) mm, rotated rx 180 ry 0 rz -179 deg; joints [-1.172, -76.207, 123.35, -1.598, -47.155, 1.087] to (-64.86, 537.16, -8.35) mm, rotated rx 180 ry 0 rz -179 deg; joints [-1.798, -76.919, 124.274, -2.444, -47.382, 1.655]
  MoveL 1640 to (-90.26, 537.16, -8.35) mm, rotated rx -180 ry 0 rz -179 deg; joints [-1.858, -78.417, 126.185, -2.509, -47.795, 1.686]
  MoveL 1641 to (-166.46, 537.16, -8.35) mm, rotated rx -180 ry 0 rz -179 deg; joints [-2.056, -83.024, 131.756, -2.734, -48.765, 1.803]
  MoveC 1642 to (-179.16, 524.46, -8.35) mm, rotated rx 180 ry 0 rz -179 deg; joints [-1.425, -83.849, 132.705, -1.891, -48.872, 1.244] to (-191.86, 537.16, -8.35) mm, rotated rx -180 ry 0 rz -179 deg; joints [-2.128, -84.605, 133.561, -2.82, -48.99, 1.851]
  MoveL 1643 to (-293.46, 537.16, -8.35) mm, rotated rx -180 ry 0 rz -179 deg; joints [-2.453, -91.256, 140.527, -3.236, -49.317, 2.11]
  MoveC 1644 to (-306.16, 524.46, -8.35) mm, rotated rx -180 ry 0 rz -179 deg; joints [-1.744, -92.18, 141.415, -2.302, -49.258, 1.503] to (-318.86, 537.16, -8.35) mm, rotated rx -180 ry 0 rz -179 deg; joints [-2.545, -93.02, 142.205, -3.361, -49.234, 2.196]
  MoveL 1645 to (-395.06, 537.16, -8.35) mm, rotated rx 180 ry 0 rz -179 deg; joints [-2.854, -98.635, 147.073, -3.812, -48.502, 2.528]
  MoveL 1646 to (-420.46, 537.16, -8.35) mm, rotated rx -180 ry 0 rz -179 deg; joints [-2.969, -100.634, 148.638, -3.992, -48.073, 2.67]
  MoveC 1647 to (-433.16, 524.46, -8.35) mm, rotated rx -180 ry 0 rz -179 deg; joints [-2.161, -101.727, 149.457, -2.919, -47.767, 1.963] to (-445.86, 537.16, -8.35) mm, rotated rx -180 ry 0 rz -179 deg; joints [-3.091, -102.71, 150.172, -4.192, -47.539, 2.833]
  MoveL 1648 to (-471.26, 537.16, -8.35) mm, rotated rx -180 ry 0 rz -179 deg; joints [-3.221, -104.869, 151.673, -4.414, -46.888, 3.02]
  MoveL 1649 to (-471.26, 384.76, -8.35) mm, rotated rx -180 ry 0 rz -179 deg; joints [7.7, -104.582, 151.478, 10.492, -47.378, -7.148]
  MoveL 1650 to (-14.06, 384.76, -8.35) mm, rotated rx -180 ry 0 rz -179 deg; joints [5.269, -73.838, 120.202, 7.262, -46.595, -5.004]
  MoveC 1651 to (-13.61, 384.57, -8.35) mm, rotated rx -180 ry 0 rz -179 deg; joints [5.276, -73.812, 120.166, 7.272, -46.586, -5.012] to (-13.42, 384.12, -8.35) mm, rotated rx -180 ry 0 rz -179 deg; joints [5.296, -73.799, 120.149, 7.3, -46.583, -5.032]
  MoveL 1652 to (-13.42, 383.49, -8.35) mm, rotated rx -180 ry 0 rz -179 deg; joints [5.324, -73.796, 120.145, 7.339, -46.585, -5.059]
  MoveC 1653 to (-13.42, 383.04, -8.16) mm, rotated rx -180 ry 0 rz -179 deg; joints [5.345, -73.802, 120.138, 7.369, -46.573, -5.081] to (-13.42, 382.85, -7.72) mm, rotated rx -180 ry 0 rz -179 deg; joints [5.353, -73.82, 120.124, 7.385, -46.542, -5.094]
  Set speed (500.0 mm/s)
  MoveL 1654 to (-13.42, 382.85, 15) mm, rotated rx -180 ry 0 rz -179 deg; joints [5.353, -74.765, 119.469, 7.588, -44.957, -5.385]
  MoveL 1655 to (-13.42, 382.85, 15) mm, rotated rx -180 ry 0 rz -179 deg; joints [5.353, -74.765, 119.469, 7.588, -44.957, -5.385]

--- program Prog2 (robot GIGASHEEN) ---
  MoveJ (plywood back right safe)
  MoveL (plywood back left safe)
  MoveL (plywood front left safe)
  MoveL (plywood front right safe)
